REGION Network 3: ANGLE CODE READING
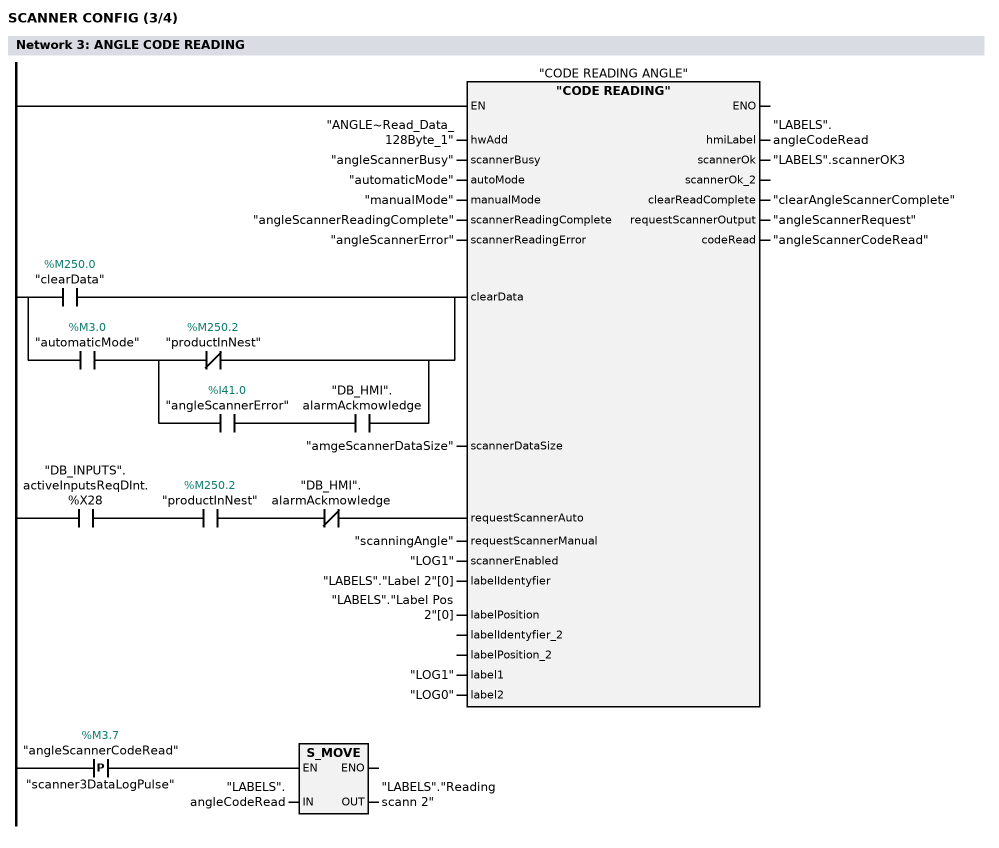
   RUNG wire#powerrail
      "CODE READING ANGLE"(clearData := wire#w2, requestScannerAuto := wire#w3, hwAdd := "ANGLE~Read_Data_128Byte_1", scannerBusy := "angleScannerBusy", autoMode := "automaticMode", manualMode := "manualMode", scannerReadingComplete := "angleScannerReadingComplete", scannerReadingError := "angleScannerError", scannerDataSize := "amgeScannerDataSize", requestScannerManual := "scanningAngle", scannerEnabled := "LOG1", labelIdentyfier := "LABELS"."Label 2"[0], labelPosition := "LABELS"."Label Pos 2"[0], labelIdentyfier_2 :=, labelPosition_2 :=, label1 := "LOG1", label2 := "LOG0", hmiLabel => "LABELS".angleCodeRead, scannerOk => "LABELS".scannerOK3, scannerOk_2 =>, clearReadComplete => "clearAngleScannerComplete", requestScannerOutput => "angleScannerRequest", codeRead => "angleScannerCodeRead")
   END_RUNG
   RUNG wire#powerrail
      Contact( "clearData" )
   END_RUNG wire#w2
   RUNG wire#powerrail
      Contact( "automaticMode" )
      wire#w1
      I_Contact( "productInNest" )
   END_RUNG wire#w2
   RUNG wire#w1
      Contact( "angleScannerError" )
      Contact( "DB_HMI".alarmAckmowledge )
   END_RUNG wire#w2
   RUNG wire#powerrail
      Contact( "DB_INPUTS".activeInputsReqDInt.%X28 )
      Contact( "productInNest" )
      I_Contact( "DB_HMI".alarmAckmowledge )
   END_RUNG wire#w3
   RUNG wire#powerrail
      P_Contact(operand := "angleScannerCodeRead", bit := "scanner3DataLogPulse")
      S_Move(in := "LABELS".angleCodeRead, out => "LABELS"."Reading scann 2")
   END_RUNG
   // the same network as SCL:
   "CODE READING ANGLE"(hwAdd := "ANGLE~Read_Data_128Byte_1",   // "CODE READING"
                        scannerBusy := "angleScannerBusy",
                        autoMode := "automaticMode",
                        manualMode := "manualMode",
                        scannerReadingComplete := "angleScannerReadingComplete",
                        scannerReadingError := "angleScannerError",
                        clearData := "clearData" OR ("automaticMode" AND (NOT "productInNest" OR ("angleScannerError" AND "DB_HMI".alarmAckmowledge))),
                        scannerDataSize := "amgeScannerDataSize",
                        requestScannerAuto := "DB_INPUTS".activeInputsReqDInt.%X28 AND "productInNest" AND NOT "DB_HMI".alarmAckmowledge,
                        requestScannerManual := "scanningAngle",
                        scannerEnabled := "LOG1",
                        labelIdentyfier := "LABELS"."Label 2"[0],
                        labelPosition := "LABELS"."Label Pos 2"[0],
                        label1 := "LOG1",
                        label2 := "LOG0",
                        hmiLabel => "LABELS".angleCodeRead,
                        scannerOk => "LABELS".scannerOK3,
                        clearReadComplete => "clearAngleScannerComplete",
                        requestScannerOutput => "angleScannerRequest",
                        codeRead => "angleScannerCodeRead");
   #_w1 := "angleScannerCodeRead" AND NOT "scanner3DataLogPulse";   // rising edge of "angleScannerCodeRead"
   "scanner3DataLogPulse" := "angleScannerCodeRead";
   IF #_w1 THEN "LABELS"."Reading scann 2" := "LABELS".angleCodeRead; END_IF;
END_REGION

REGION Network 4: Move values to HMI
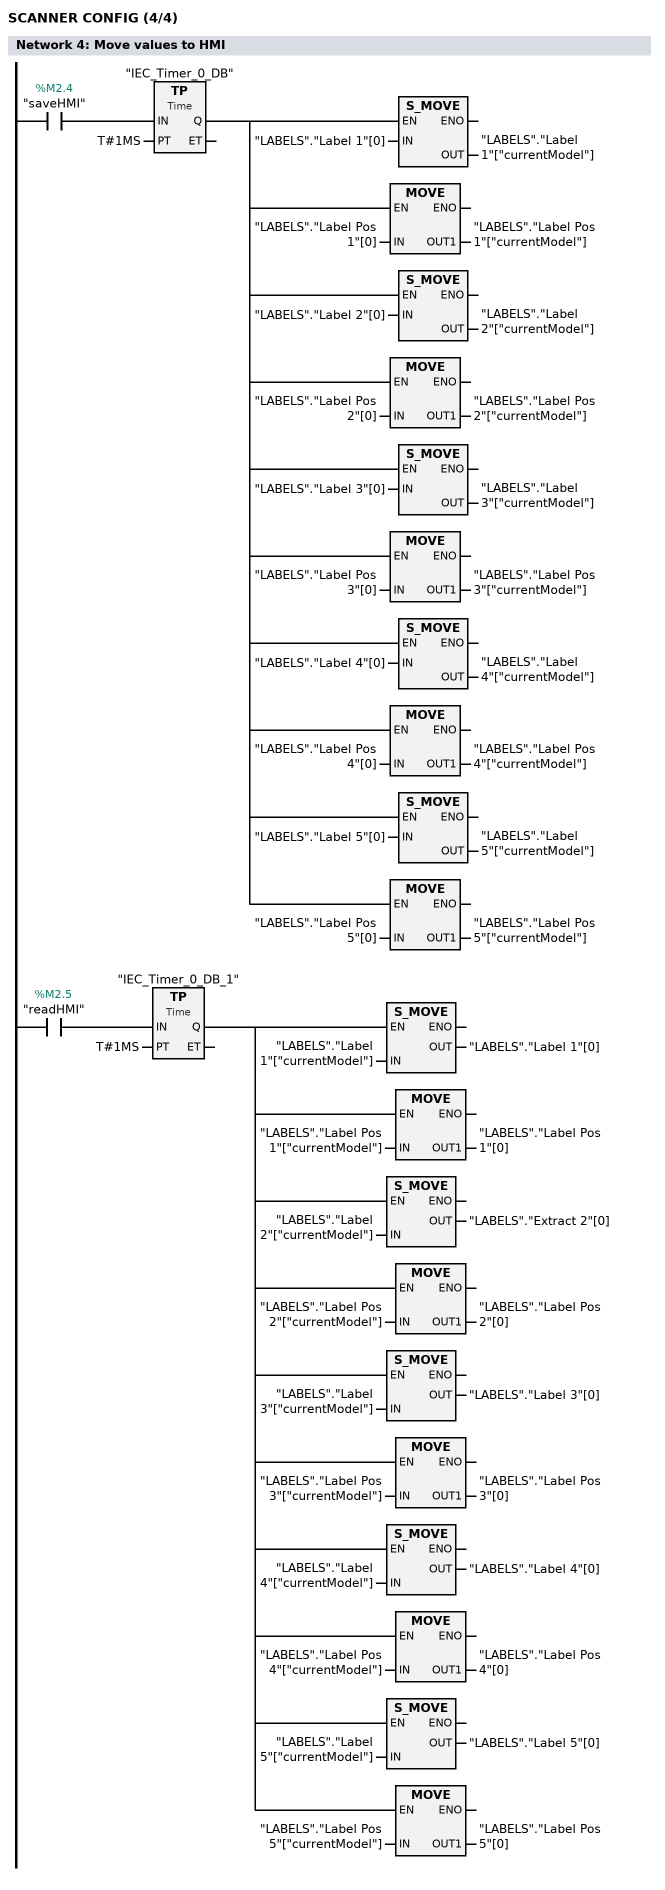
   RUNG wire#powerrail
      Contact( "saveHMI" )
      { S7_Templates := "time_type := Time" } "IEC_Timer_0_DB".TP(pt := T#1MS, et =>)
      wire#w1
      S_Move(in := "LABELS"."Label 1"[0], out => "LABELS"."Label 1"["currentModel"])
   END_RUNG
   RUNG wire#w1
      Move(in := "LABELS"."Label Pos 1"[0], out1 => "LABELS"."Label Pos 1"["currentModel"])
   END_RUNG
   RUNG wire#w1
      S_Move(in := "LABELS"."Label 2"[0], out => "LABELS"."Label 2"["currentModel"])
   END_RUNG
   RUNG wire#w1
      Move(in := "LABELS"."Label Pos 2"[0], out1 => "LABELS"."Label Pos 2"["currentModel"])
   END_RUNG
   RUNG wire#w1
      S_Move(in := "LABELS"."Label 3"[0], out => "LABELS"."Label 3"["currentModel"])
   END_RUNG
   RUNG wire#w1
      Move(in := "LABELS"."Label Pos 3"[0], out1 => "LABELS"."Label Pos 3"["currentModel"])
   END_RUNG
   RUNG wire#w1
      S_Move(in := "LABELS"."Label 4"[0], out => "LABELS"."Label 4"["currentModel"])
   END_RUNG
   RUNG wire#w1
      Move(in := "LABELS"."Label Pos 4"[0], out1 => "LABELS"."Label Pos 4"["currentModel"])
   END_RUNG
   RUNG wire#w1
      S_Move(in := "LABELS"."Label 5"[0], out => "LABELS"."Label 5"["currentModel"])
   END_RUNG
   RUNG wire#w1
      Move(in := "LABELS"."Label Pos 5"[0], out1 => "LABELS"."Label Pos 5"["currentModel"])
   END_RUNG
   RUNG wire#powerrail
      Contact( "readHMI" )
      { S7_Templates := "time_type := Time" } "IEC_Timer_0_DB_1".TP(pt := T#1MS, et =>)
      wire#w2
      S_Move(in := "LABELS"."Label 1"["currentModel"], out => "LABELS"."Label 1"[0])
   END_RUNG
   RUNG wire#w2
      Move(in := "LABELS"."Label Pos 1"["currentModel"], out1 => "LABELS"."Label Pos 1"[0])
   END_RUNG
   RUNG wire#w2
      S_Move(in := "LABELS"."Label 2"["currentModel"], out => "LABELS"."Extract 2"[0])
   END_RUNG
   RUNG wire#w2
      Move(in := "LABELS"."Label Pos 2"["currentModel"], out1 => "LABELS"."Label Pos 2"[0])
   END_RUNG
   RUNG wire#w2
      S_Move(in := "LABELS"."Label 3"["currentModel"], out => "LABELS"."Label 3"[0])
   END_RUNG
   RUNG wire#w2
      Move(in := "LABELS"."Label Pos 3"["currentModel"], out1 => "LABELS"."Label Pos 3"[0])
   END_RUNG
   RUNG wire#w2
      S_Move(in := "LABELS"."Label 4"["currentModel"], out => "LABELS"."Label 4"[0])
   END_RUNG
   RUNG wire#w2
      Move(in := "LABELS"."Label Pos 4"["currentModel"], out1 => "LABELS"."Label Pos 4"[0])
   END_RUNG
   RUNG wire#w2
      S_Move(in := "LABELS"."Label 5"["currentModel"], out => "LABELS"."Label 5"[0])
   END_RUNG
   RUNG wire#w2
      Move(in := "LABELS"."Label Pos 5"["currentModel"], out1 => "LABELS"."Label Pos 5"[0])
   END_RUNG
   // the same network as SCL:
   "IEC_Timer_0_DB".TP(IN := "saveHMI", PT := T#1MS);
   IF "IEC_Timer_0_DB".Q THEN
       "LABELS"."Label 1"["currentModel"] := "LABELS"."Label 1"[0];
       "LABELS"."Label Pos 1"["currentModel"] := "LABELS"."Label Pos 1"[0];
       "LABELS"."Label 2"["currentModel"] := "LABELS"."Label 2"[0];
       "LABELS"."Label Pos 2"["currentModel"] := "LABELS"."Label Pos 2"[0];
       "LABELS"."Label 3"["currentModel"] := "LABELS"."Label 3"[0];
       "LABELS"."Label Pos 3"["currentModel"] := "LABELS"."Label Pos 3"[0];
       "LABELS"."Label 4"["currentModel"] := "LABELS"."Label 4"[0];
       "LABELS"."Label Pos 4"["currentModel"] := "LABELS"."Label Pos 4"[0];
       "LABELS"."Label 5"["currentModel"] := "LABELS"."Label 5"[0];
       "LABELS"."Label Pos 5"["currentModel"] := "LABELS"."Label Pos 5"[0];
   END_IF;
   "IEC_Timer_0_DB_1".TP(IN := "readHMI", PT := T#1MS);
   IF "IEC_Timer_0_DB_1".Q THEN
       "LABELS"."Label 1"[0] := "LABELS"."Label 1"["currentModel"];
       "LABELS"."Label Pos 1"[0] := "LABELS"."Label Pos 1"["currentModel"];
       "LABELS"."Extract 2"[0] := "LABELS"."Label 2"["currentModel"];
       "LABELS"."Label Pos 2"[0] := "LABELS"."Label Pos 2"["currentModel"];
       "LABELS"."Label 3"[0] := "LABELS"."Label 3"["currentModel"];
       "LABELS"."Label Pos 3"[0] := "LABELS"."Label Pos 3"["currentModel"];
       "LABELS"."Label 4"[0] := "LABELS"."Label 4"["currentModel"];
       "LABELS"."Label Pos 4"[0] := "LABELS"."Label Pos 4"["currentModel"];
       "LABELS"."Label 5"[0] := "LABELS"."Label 5"["currentModel"];
       "LABELS"."Label Pos 5"[0] := "LABELS"."Label Pos 5"["currentModel"];
   END_IF;
END_REGION
END_FUNCTION

FUNCTION_BLOCK "CODE READING"   // FB13, LAD
{ S7_Optimized_Access := 'TRUE' }
VERSION : 0.1
// stored: AutoNumber true, IsIECCheckEnabled false, IsRetainMemResEnabled false, MemoryReserve 100, SetENOAutomatically false, UDAEnableTagReadback false
   VAR_INPUT
      hwAdd : HW_IO;
      scannerBusy : Bool;
      autoMode : Bool;
      manualMode : Bool;
      scannerReadingComplete : Bool;
      scannerReadingError : Bool;
      clearData : Bool;
      scannerDataSize : Int;
      requestScannerAuto : Bool;
      requestScannerManual : Bool;
      scannerEnabled : Bool;
      labelIdentyfier : String[5];
      labelPosition : Int;
      labelIdentyfier_2 : String[5];
      labelPosition_2 : Int;
      label1 : Bool;
      label2 : Bool;
   END_VAR
   VAR_OUTPUT
      hmiLabel : String[180];
      scannerOk : Bool;
      scannerOk_2 : Bool;
      clearReadComplete : Bool;
      requestScannerOutput : Bool;
      codeRead : Bool;
   END_VAR
   VAR
      scannerReading { ExternalAccessible := 'False'; ExternalVisible := 'False'; ExternalWritable := 'False'} : Array[0..254] of Char;
      ScannerReadTimer { S7_SetPoint := 'True'} : TON_TIME;
   END_VAR
   VAR_TEMP
      scannerError : Int;
      receiveCode : String[80];
      readingScann1 : String[180];
      scannerLength : Int;
      labelExtract : String[10];
   END_VAR
   VAR_TEMP   // added for the SCL form of the ladder/FBD networks
      _w1 : Bool;
      _w2 : Bool;
      _w3 : Bool;
      _w4 : Bool;
      _w5 : Bool;
      _w6 : Bool;
      _w7 : Bool;
      _w8 : Bool;
      _w9 : Bool;
      _w10 : Bool;
      _w11 : Bool;
   END_VAR
BEGIN

REGION Network 1: REQUEST SCANNER
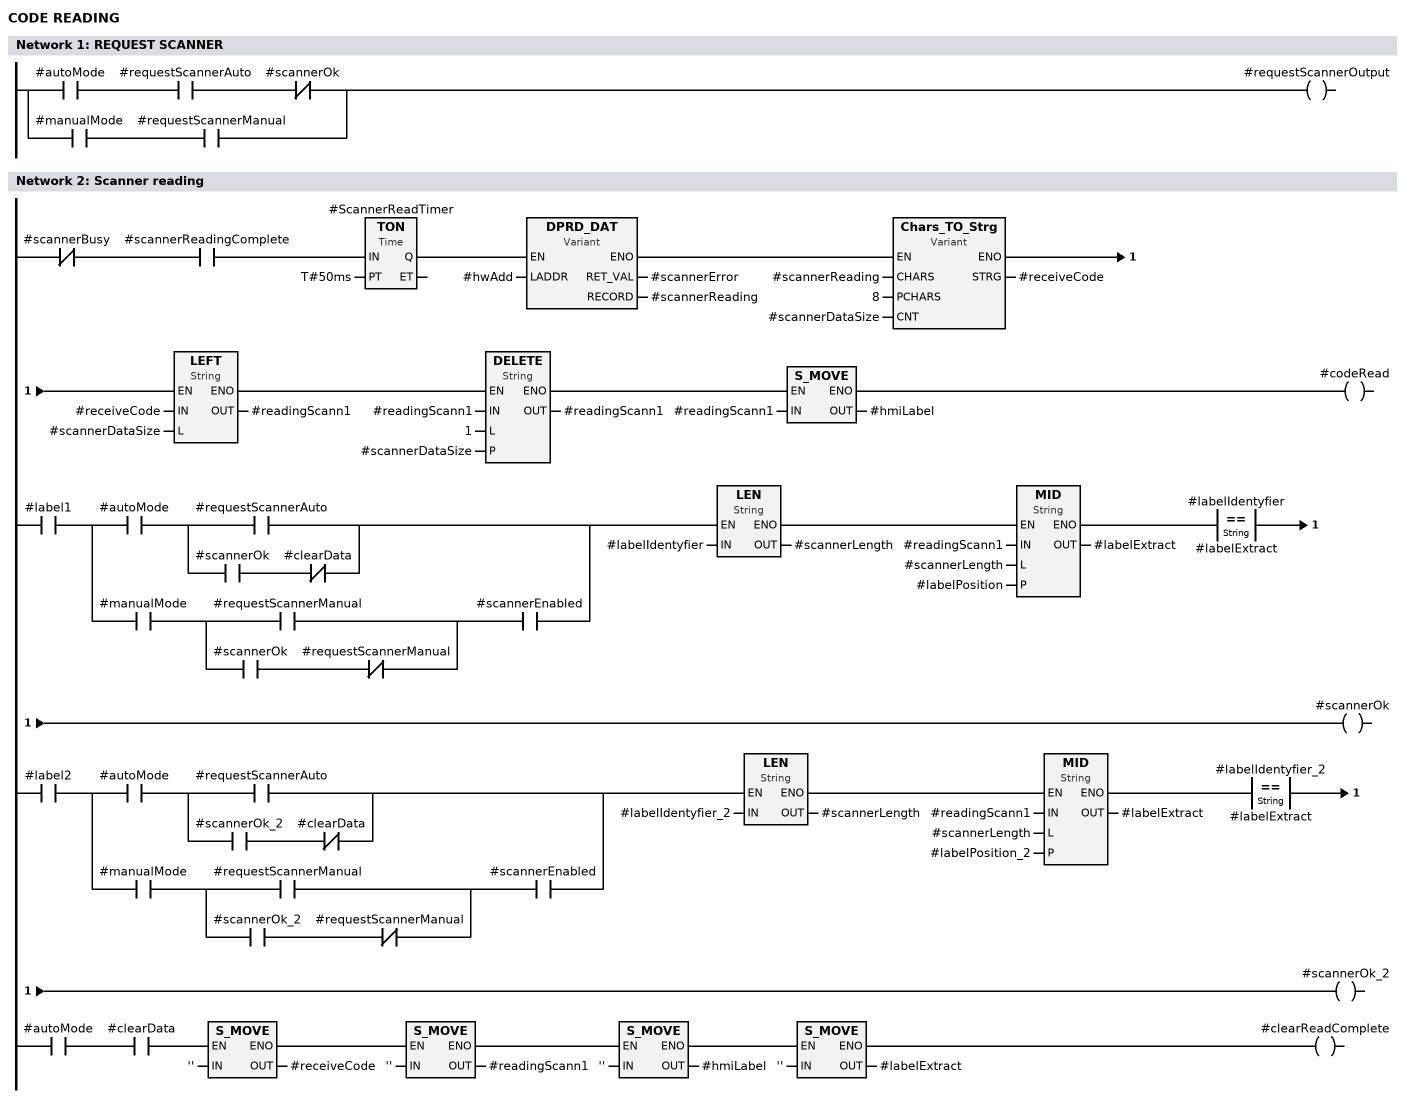
   RUNG wire#powerrail
      Contact( #autoMode )
      Contact( #requestScannerAuto )
      I_Contact( #scannerOk )
      wire#w1
      Coil( #requestScannerOutput )
   END_RUNG
   RUNG wire#powerrail
      Contact( #manualMode )
      Contact( #requestScannerManual )
   END_RUNG wire#w1
   // the same network as SCL:
   #requestScannerOutput := (#autoMode AND #requestScannerAuto AND NOT #scannerOk) OR (#manualMode AND #requestScannerManual);
END_REGION

REGION Network 2: Scanner reading
   RUNG wire#powerrail
      I_Contact( #scannerBusy )
      Contact( #scannerReadingComplete )
      { S7_Templates := "time_type := Time" } #ScannerReadTimer.TON(pt := T#50ms, et =>)
      { S7_Templates := "[ptr_type := Variant, laddr_type := HW_IO]" } DPRD_DAT(LADDR := #hwAdd, RET_VAL => #scannerError, RECORD => #scannerReading)
      { S7_Templates := "[ptr_type := Variant, str_type := String]" } Chars_TO_Strg(Chars := #scannerReading, pChars := 8, Cnt := #scannerDataSize, Strg => #receiveCode)
      { S7_Templates := "str_type := String" } LEFT(IN := #receiveCode, L := #scannerDataSize, OUT => #readingScann1)
      { S7_Templates := "str_type := String" } DELETE(IN := #readingScann1, L := 1, P := #scannerDataSize, OUT => #readingScann1)
      S_Move(in := #readingScann1, out => #hmiLabel)
      Coil( #codeRead )
   END_RUNG
   RUNG wire#powerrail
      Contact( #label1 )
      wire#w1
      Contact( #autoMode )
      wire#w2
      Contact( #requestScannerAuto )
      wire#w3
      { S7_Templates := "[str_type := String, return_type := Int]" } LEN(IN := #labelIdentyfier, OUT => #scannerLength)
      { S7_Templates := "value_type := String" } MID(IN := #readingScann1, L := #scannerLength, P := #labelPosition, OUT => #labelExtract)
      { S7_Templates := "SrcType := String" } EQ_Contact(in1 := #labelIdentyfier, in2 := #labelExtract)
      Coil( #scannerOk )
   END_RUNG
   RUNG wire#w2
      Contact( #scannerOk )
      I_Contact( #clearData )
   END_RUNG wire#w3
   RUNG wire#w1
      Contact( #manualMode )
      wire#w4
      Contact( #requestScannerManual )
      wire#w5
      Contact( #scannerEnabled )
   END_RUNG wire#w3
   RUNG wire#w4
      Contact( #scannerOk )
      I_Contact( #requestScannerManual )
   END_RUNG wire#w5
   RUNG wire#powerrail
      Contact( #label2 )
      wire#w6
      Contact( #autoMode )
      wire#w7
      Contact( #requestScannerAuto )
      wire#w8
      { S7_Templates := "[str_type := String, return_type := Int]" } LEN(IN := #labelIdentyfier_2, OUT => #scannerLength)
      { S7_Templates := "value_type := String" } MID(IN := #readingScann1, L := #scannerLength, P := #labelPosition_2, OUT => #labelExtract)
      { S7_Templates := "SrcType := String" } EQ_Contact(in1 := #labelIdentyfier_2, in2 := #labelExtract)
      Coil( #scannerOk_2 )
   END_RUNG
   RUNG wire#w7
      Contact( #scannerOk_2 )
      I_Contact( #clearData )
   END_RUNG wire#w8
   RUNG wire#w6
      Contact( #manualMode )
      wire#w9
      Contact( #requestScannerManual )
      wire#w10
      Contact( #scannerEnabled )
   END_RUNG wire#w8
   RUNG wire#w9
      Contact( #scannerOk_2 )
      I_Contact( #requestScannerManual )
   END_RUNG wire#w10
   RUNG wire#powerrail
      Contact( #autoMode )
      Contact( #clearData )
      S_Move(in := '', out => #receiveCode)
      S_Move(in := '', out => #readingScann1)
      S_Move(in := '', out => #hmiLabel)
      S_Move(in := '', out => #labelExtract)
      Coil( #clearReadComplete )
   END_RUNG
   // the same network as SCL:
   #ScannerReadTimer(IN := NOT #scannerBusy AND #scannerReadingComplete, PT := T#50ms);   // TON
   #scannerError := DPRD_DAT(EN := #ScannerReadTimer.Q, LADDR := #hwAdd, RECORD => #scannerReading, ENO => #_w1);
   Chars_TO_Strg(EN := #_w1,
                 Chars := #scannerReading,
                 pChars := 8,
                 Cnt := #scannerDataSize,
                 Strg => #receiveCode,
                 ENO => #_w2);
   LEFT(EN := #_w2, IN := #receiveCode, L := #scannerDataSize, OUT => #readingScann1, ENO => #_w3);
   DELETE(EN := #_w3, IN := #readingScann1, L := 1, P := #scannerDataSize, OUT => #readingScann1, ENO => #_w4);
   IF #_w4 THEN #hmiLabel := #readingScann1; END_IF;
   #codeRead := #_w4;
   #_w5 := #label1 AND ((#autoMode AND (#requestScannerAuto OR (#scannerOk AND NOT #clearData))) OR (#manualMode AND (#requestScannerManual OR (#scannerOk AND NOT #requestScannerManual)) AND #scannerEnabled));
   LEN(EN := #_w5, IN := #labelIdentyfier, OUT => #scannerLength, ENO => #_w6);
   MID(EN := #_w6,
       IN := #readingScann1,
       L := #scannerLength,
       P := #labelPosition,
       OUT => #labelExtract,
       ENO => #_w7);
   #scannerOk := #_w7 AND (#labelIdentyfier = #labelExtract);
   #_w8 := #label2 AND ((#autoMode AND (#requestScannerAuto OR (#scannerOk_2 AND NOT #clearData))) OR (#manualMode AND (#requestScannerManual OR (#scannerOk_2 AND NOT #requestScannerManual)) AND #scannerEnabled));
   LEN(EN := #_w8, IN := #labelIdentyfier_2, OUT => #scannerLength, ENO => #_w9);
   MID(EN := #_w9,
       IN := #readingScann1,
       L := #scannerLength,
       P := #labelPosition_2,
       OUT => #labelExtract,
       ENO => #_w10);
   #scannerOk_2 := #_w10 AND (#labelIdentyfier_2 = #labelExtract);
   #_w11 := #autoMode AND #clearData;
   IF #_w11 THEN
       #receiveCode := '';
       #readingScann1 := '';
       #hmiLabel := '';
       #labelExtract := '';
   END_IF;
   #clearReadComplete := #_w11;
END_REGION
END_FUNCTION_BLOCK

FUNCTION "DINT TO BOOL" : Void   // FC10, LAD
{ S7_Optimized_Access := 'TRUE' }
VERSION : 0.1
// stored: AutoNumber true, IsIECCheckEnabled false, SetENOAutomatically false, UDAEnableTagReadback false
BEGIN

REGION Network 1: A INPUTS STATUS
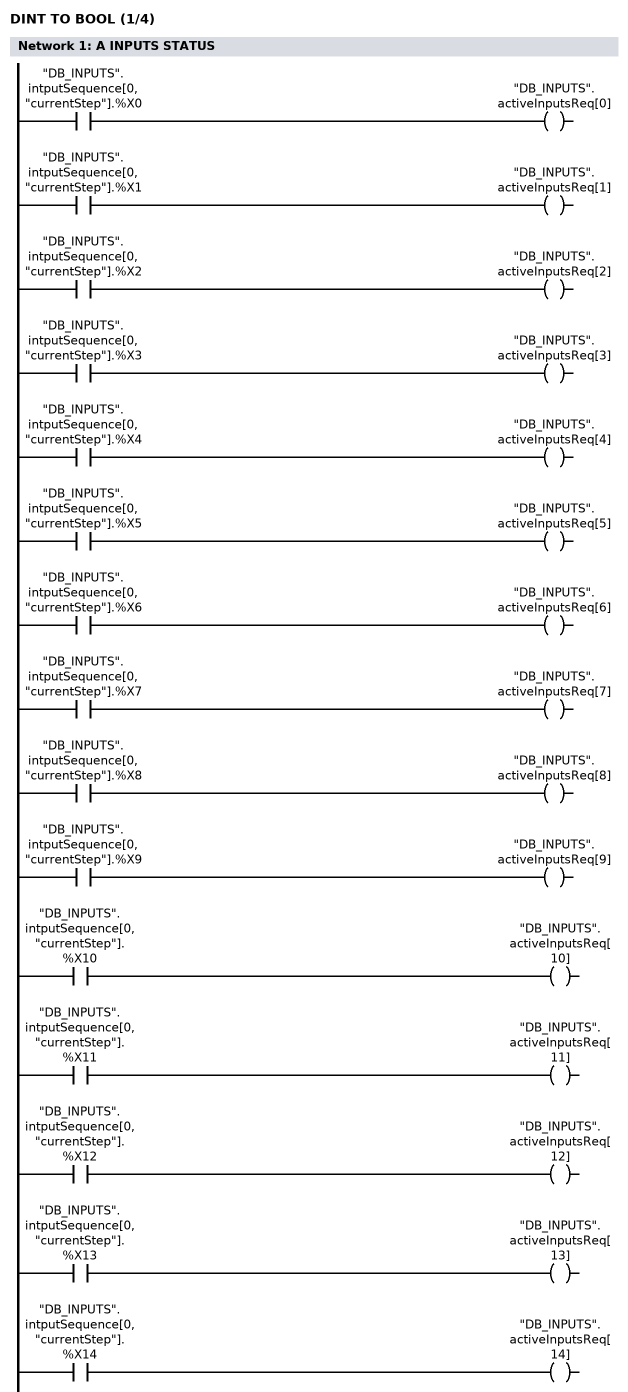
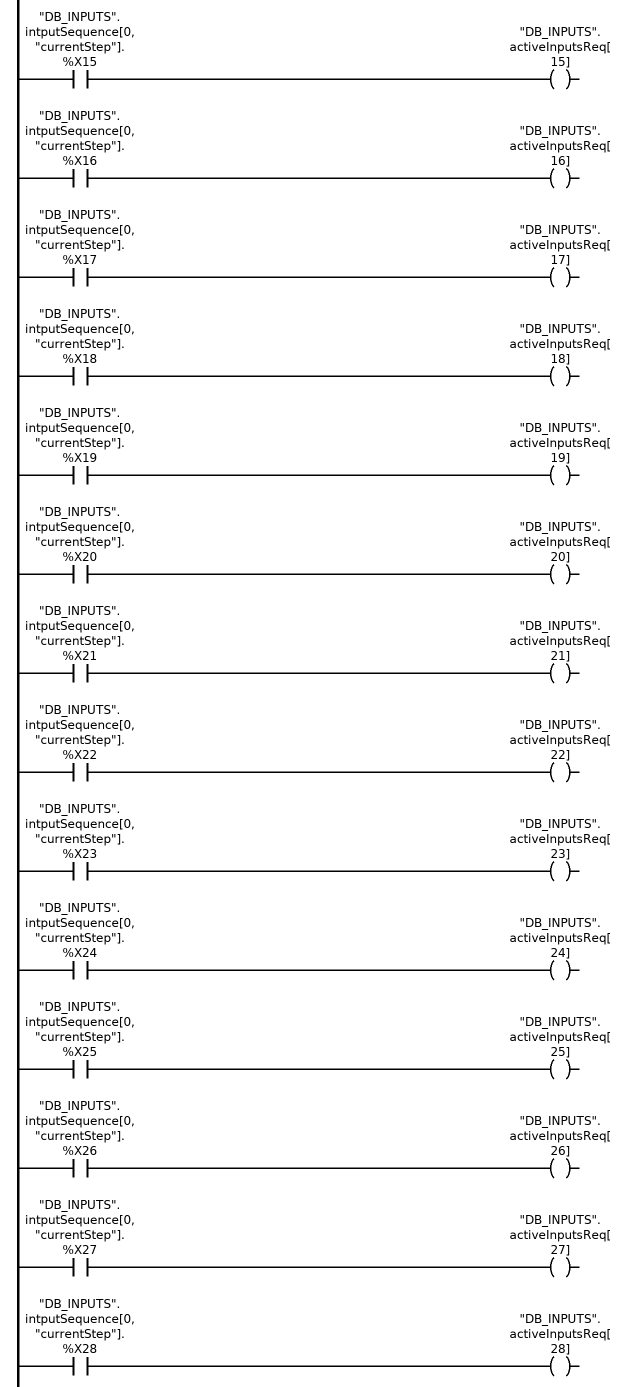
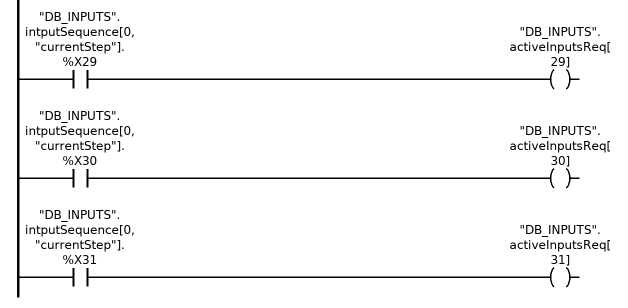
   RUNG wire#powerrail
      Contact( "DB_INPUTS".intputSequence[0, "currentStep"].%X0 )
      Coil( "DB_INPUTS".activeInputsReq[0] )
   END_RUNG
   RUNG wire#powerrail
      Contact( "DB_INPUTS".intputSequence[0, "currentStep"].%X1 )
      Coil( "DB_INPUTS".activeInputsReq[1] )
   END_RUNG
   RUNG wire#powerrail
      Contact( "DB_INPUTS".intputSequence[0, "currentStep"].%X2 )
      Coil( "DB_INPUTS".activeInputsReq[2] )
   END_RUNG
   RUNG wire#powerrail
      Contact( "DB_INPUTS".intputSequence[0, "currentStep"].%X3 )
      Coil( "DB_INPUTS".activeInputsReq[3] )
   END_RUNG
   RUNG wire#powerrail
      Contact( "DB_INPUTS".intputSequence[0, "currentStep"].%X4 )
      Coil( "DB_INPUTS".activeInputsReq[4] )
   END_RUNG
   RUNG wire#powerrail
      Contact( "DB_INPUTS".intputSequence[0, "currentStep"].%X5 )
      Coil( "DB_INPUTS".activeInputsReq[5] )
   END_RUNG
   RUNG wire#powerrail
      Contact( "DB_INPUTS".intputSequence[0, "currentStep"].%X6 )
      Coil( "DB_INPUTS".activeInputsReq[6] )
   END_RUNG
   RUNG wire#powerrail
      Contact( "DB_INPUTS".intputSequence[0, "currentStep"].%X7 )
      Coil( "DB_INPUTS".activeInputsReq[7] )
   END_RUNG
   RUNG wire#powerrail
      Contact( "DB_INPUTS".intputSequence[0, "currentStep"].%X8 )
      Coil( "DB_INPUTS".activeInputsReq[8] )
   END_RUNG
   RUNG wire#powerrail
      Contact( "DB_INPUTS".intputSequence[0, "currentStep"].%X9 )
      Coil( "DB_INPUTS".activeInputsReq[9] )
   END_RUNG
   RUNG wire#powerrail
      Contact( "DB_INPUTS".intputSequence[0, "currentStep"].%X10 )
      Coil( "DB_INPUTS".activeInputsReq[10] )
   END_RUNG
   RUNG wire#powerrail
      Contact( "DB_INPUTS".intputSequence[0, "currentStep"].%X11 )
      Coil( "DB_INPUTS".activeInputsReq[11] )
   END_RUNG
   RUNG wire#powerrail
      Contact( "DB_INPUTS".intputSequence[0, "currentStep"].%X12 )
      Coil( "DB_INPUTS".activeInputsReq[12] )
   END_RUNG
   RUNG wire#powerrail
      Contact( "DB_INPUTS".intputSequence[0, "currentStep"].%X13 )
      Coil( "DB_INPUTS".activeInputsReq[13] )
   END_RUNG
   RUNG wire#powerrail
      Contact( "DB_INPUTS".intputSequence[0, "currentStep"].%X14 )
      Coil( "DB_INPUTS".activeInputsReq[14] )
   END_RUNG
   RUNG wire#powerrail
      Contact( "DB_INPUTS".intputSequence[0, "currentStep"].%X15 )
      Coil( "DB_INPUTS".activeInputsReq[15] )
   END_RUNG
   RUNG wire#powerrail
      Contact( "DB_INPUTS".intputSequence[0, "currentStep"].%X16 )
      Coil( "DB_INPUTS".activeInputsReq[16] )
   END_RUNG
   RUNG wire#powerrail
      Contact( "DB_INPUTS".intputSequence[0, "currentStep"].%X17 )
      Coil( "DB_INPUTS".activeInputsReq[17] )
   END_RUNG
   RUNG wire#powerrail
      Contact( "DB_INPUTS".intputSequence[0, "currentStep"].%X18 )
      Coil( "DB_INPUTS".activeInputsReq[18] )
   END_RUNG
   RUNG wire#powerrail
      Contact( "DB_INPUTS".intputSequence[0, "currentStep"].%X19 )
      Coil( "DB_INPUTS".activeInputsReq[19] )
   END_RUNG
   RUNG wire#powerrail
      Contact( "DB_INPUTS".intputSequence[0, "currentStep"].%X20 )
      Coil( "DB_INPUTS".activeInputsReq[20] )
   END_RUNG
   RUNG wire#powerrail
      Contact( "DB_INPUTS".intputSequence[0, "currentStep"].%X21 )
      Coil( "DB_INPUTS".activeInputsReq[21] )
   END_RUNG
   RUNG wire#powerrail
      Contact( "DB_INPUTS".intputSequence[0, "currentStep"].%X22 )
      Coil( "DB_INPUTS".activeInputsReq[22] )
   END_RUNG
   RUNG wire#powerrail
      Contact( "DB_INPUTS".intputSequence[0, "currentStep"].%X23 )
      Coil( "DB_INPUTS".activeInputsReq[23] )
   END_RUNG
   RUNG wire#powerrail
      Contact( "DB_INPUTS".intputSequence[0, "currentStep"].%X24 )
      Coil( "DB_INPUTS".activeInputsReq[24] )
   END_RUNG
   RUNG wire#powerrail
      Contact( "DB_INPUTS".intputSequence[0, "currentStep"].%X25 )
      Coil( "DB_INPUTS".activeInputsReq[25] )
   END_RUNG
   RUNG wire#powerrail
      Contact( "DB_INPUTS".intputSequence[0, "currentStep"].%X26 )
      Coil( "DB_INPUTS".activeInputsReq[26] )
   END_RUNG
   RUNG wire#powerrail
      Contact( "DB_INPUTS".intputSequence[0, "currentStep"].%X27 )
      Coil( "DB_INPUTS".activeInputsReq[27] )
   END_RUNG
   RUNG wire#powerrail
      Contact( "DB_INPUTS".intputSequence[0, "currentStep"].%X28 )
      Coil( "DB_INPUTS".activeInputsReq[28] )
   END_RUNG
   RUNG wire#powerrail
      Contact( "DB_INPUTS".intputSequence[0, "currentStep"].%X29 )
      Coil( "DB_INPUTS".activeInputsReq[29] )
   END_RUNG
   RUNG wire#powerrail
      Contact( "DB_INPUTS".intputSequence[0, "currentStep"].%X30 )
      Coil( "DB_INPUTS".activeInputsReq[30] )
   END_RUNG
   RUNG wire#powerrail
      Contact( "DB_INPUTS".intputSequence[0, "currentStep"].%X31 )
      Coil( "DB_INPUTS".activeInputsReq[31] )
   END_RUNG
   // the same network as SCL:
   "DB_INPUTS".activeInputsReq[0] := "DB_INPUTS".intputSequence[0, "currentStep"].%X0;
   "DB_INPUTS".activeInputsReq[1] := "DB_INPUTS".intputSequence[0, "currentStep"].%X1;
   "DB_INPUTS".activeInputsReq[2] := "DB_INPUTS".intputSequence[0, "currentStep"].%X2;
   "DB_INPUTS".activeInputsReq[3] := "DB_INPUTS".intputSequence[0, "currentStep"].%X3;
   "DB_INPUTS".activeInputsReq[4] := "DB_INPUTS".intputSequence[0, "currentStep"].%X4;
   "DB_INPUTS".activeInputsReq[5] := "DB_INPUTS".intputSequence[0, "currentStep"].%X5;
   "DB_INPUTS".activeInputsReq[6] := "DB_INPUTS".intputSequence[0, "currentStep"].%X6;
   "DB_INPUTS".activeInputsReq[7] := "DB_INPUTS".intputSequence[0, "currentStep"].%X7;
   "DB_INPUTS".activeInputsReq[8] := "DB_INPUTS".intputSequence[0, "currentStep"].%X8;
   "DB_INPUTS".activeInputsReq[9] := "DB_INPUTS".intputSequence[0, "currentStep"].%X9;
   "DB_INPUTS".activeInputsReq[10] := "DB_INPUTS".intputSequence[0, "currentStep"].%X10;
   "DB_INPUTS".activeInputsReq[11] := "DB_INPUTS".intputSequence[0, "currentStep"].%X11;
   "DB_INPUTS".activeInputsReq[12] := "DB_INPUTS".intputSequence[0, "currentStep"].%X12;
   "DB_INPUTS".activeInputsReq[13] := "DB_INPUTS".intputSequence[0, "currentStep"].%X13;
   "DB_INPUTS".activeInputsReq[14] := "DB_INPUTS".intputSequence[0, "currentStep"].%X14;
   "DB_INPUTS".activeInputsReq[15] := "DB_INPUTS".intputSequence[0, "currentStep"].%X15;
   "DB_INPUTS".activeInputsReq[16] := "DB_INPUTS".intputSequence[0, "currentStep"].%X16;
   "DB_INPUTS".activeInputsReq[17] := "DB_INPUTS".intputSequence[0, "currentStep"].%X17;
   "DB_INPUTS".activeInputsReq[18] := "DB_INPUTS".intputSequence[0, "currentStep"].%X18;
   "DB_INPUTS".activeInputsReq[19] := "DB_INPUTS".intputSequence[0, "currentStep"].%X19;
   "DB_INPUTS".activeInputsReq[20] := "DB_INPUTS".intputSequence[0, "currentStep"].%X20;
   "DB_INPUTS".activeInputsReq[21] := "DB_INPUTS".intputSequence[0, "currentStep"].%X21;
   "DB_INPUTS".activeInputsReq[22] := "DB_INPUTS".intputSequence[0, "currentStep"].%X22;
   "DB_INPUTS".activeInputsReq[23] := "DB_INPUTS".intputSequence[0, "currentStep"].%X23;
   "DB_INPUTS".activeInputsReq[24] := "DB_INPUTS".intputSequence[0, "currentStep"].%X24;
   "DB_INPUTS".activeInputsReq[25] := "DB_INPUTS".intputSequence[0, "currentStep"].%X25;
   "DB_INPUTS".activeInputsReq[26] := "DB_INPUTS".intputSequence[0, "currentStep"].%X26;
   "DB_INPUTS".activeInputsReq[27] := "DB_INPUTS".intputSequence[0, "currentStep"].%X27;
   "DB_INPUTS".activeInputsReq[28] := "DB_INPUTS".intputSequence[0, "currentStep"].%X28;
   "DB_INPUTS".activeInputsReq[29] := "DB_INPUTS".intputSequence[0, "currentStep"].%X29;
   "DB_INPUTS".activeInputsReq[30] := "DB_INPUTS".intputSequence[0, "currentStep"].%X30;
   "DB_INPUTS".activeInputsReq[31] := "DB_INPUTS".intputSequence[0, "currentStep"].%X31;
END_REGION

REGION Network 2: MASK INPUTS STATUS
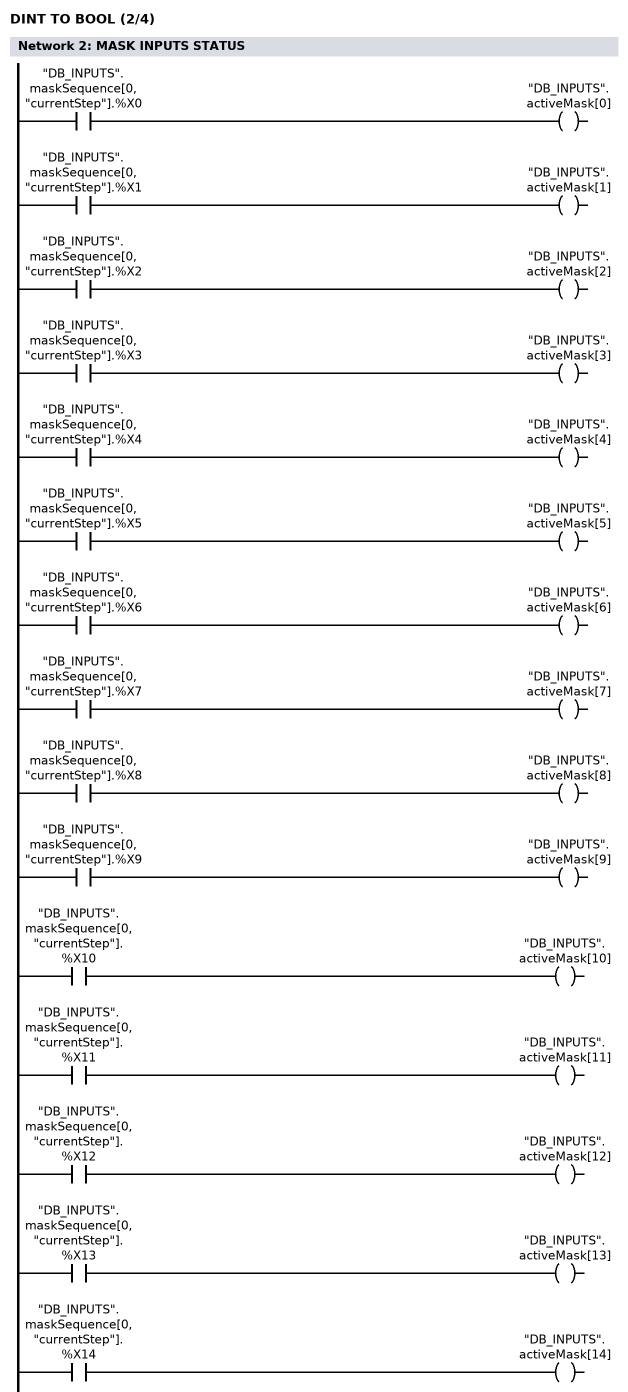
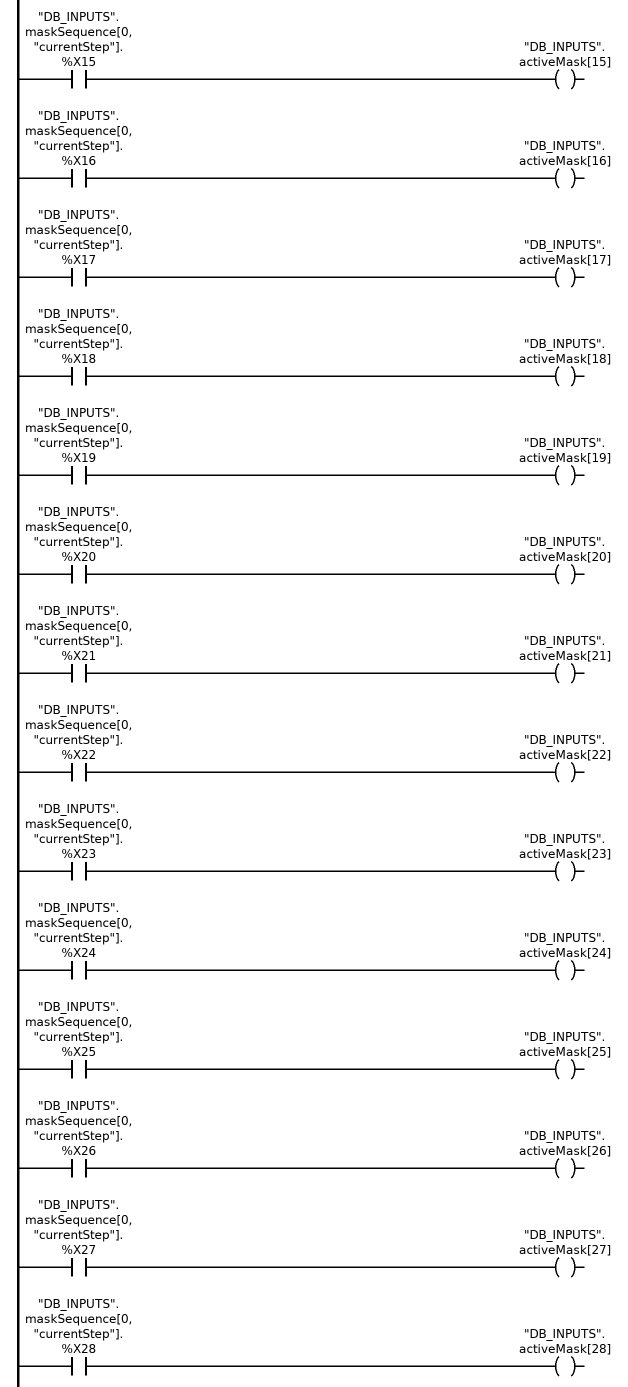
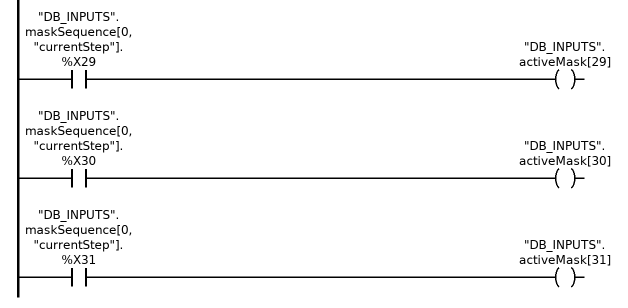
   RUNG wire#powerrail
      Contact( "DB_INPUTS".maskSequence[0, "currentStep"].%X0 )
      Coil( "DB_INPUTS".activeMask[0] )
   END_RUNG
   RUNG wire#powerrail
      Contact( "DB_INPUTS".maskSequence[0, "currentStep"].%X1 )
      Coil( "DB_INPUTS".activeMask[1] )
   END_RUNG
   RUNG wire#powerrail
      Contact( "DB_INPUTS".maskSequence[0, "currentStep"].%X2 )
      Coil( "DB_INPUTS".activeMask[2] )
   END_RUNG
   RUNG wire#powerrail
      Contact( "DB_INPUTS".maskSequence[0, "currentStep"].%X3 )
      Coil( "DB_INPUTS".activeMask[3] )
   END_RUNG
   RUNG wire#powerrail
      Contact( "DB_INPUTS".maskSequence[0, "currentStep"].%X4 )
      Coil( "DB_INPUTS".activeMask[4] )
   END_RUNG
   RUNG wire#powerrail
      Contact( "DB_INPUTS".maskSequence[0, "currentStep"].%X5 )
      Coil( "DB_INPUTS".activeMask[5] )
   END_RUNG
   RUNG wire#powerrail
      Contact( "DB_INPUTS".maskSequence[0, "currentStep"].%X6 )
      Coil( "DB_INPUTS".activeMask[6] )
   END_RUNG
   RUNG wire#powerrail
      Contact( "DB_INPUTS".maskSequence[0, "currentStep"].%X7 )
      Coil( "DB_INPUTS".activeMask[7] )
   END_RUNG
   RUNG wire#powerrail
      Contact( "DB_INPUTS".maskSequence[0, "currentStep"].%X8 )
      Coil( "DB_INPUTS".activeMask[8] )
   END_RUNG
   RUNG wire#powerrail
      Contact( "DB_INPUTS".maskSequence[0, "currentStep"].%X9 )
      Coil( "DB_INPUTS".activeMask[9] )
   END_RUNG
   RUNG wire#powerrail
      Contact( "DB_INPUTS".maskSequence[0, "currentStep"].%X10 )
      Coil( "DB_INPUTS".activeMask[10] )
   END_RUNG
   RUNG wire#powerrail
      Contact( "DB_INPUTS".maskSequence[0, "currentStep"].%X11 )
      Coil( "DB_INPUTS".activeMask[11] )
   END_RUNG
   RUNG wire#powerrail
      Contact( "DB_INPUTS".maskSequence[0, "currentStep"].%X12 )
      Coil( "DB_INPUTS".activeMask[12] )
   END_RUNG
   RUNG wire#powerrail
      Contact( "DB_INPUTS".maskSequence[0, "currentStep"].%X13 )
      Coil( "DB_INPUTS".activeMask[13] )
   END_RUNG
   RUNG wire#powerrail
      Contact( "DB_INPUTS".maskSequence[0, "currentStep"].%X14 )
      Coil( "DB_INPUTS".activeMask[14] )
   END_RUNG
   RUNG wire#powerrail
      Contact( "DB_INPUTS".maskSequence[0, "currentStep"].%X15 )
      Coil( "DB_INPUTS".activeMask[15] )
   END_RUNG
   RUNG wire#powerrail
      Contact( "DB_INPUTS".maskSequence[0, "currentStep"].%X16 )
      Coil( "DB_INPUTS".activeMask[16] )
   END_RUNG
   RUNG wire#powerrail
      Contact( "DB_INPUTS".maskSequence[0, "currentStep"].%X17 )
      Coil( "DB_INPUTS".activeMask[17] )
   END_RUNG
   RUNG wire#powerrail
      Contact( "DB_INPUTS".maskSequence[0, "currentStep"].%X18 )
      Coil( "DB_INPUTS".activeMask[18] )
   END_RUNG
   RUNG wire#powerrail
      Contact( "DB_INPUTS".maskSequence[0, "currentStep"].%X19 )
      Coil( "DB_INPUTS".activeMask[19] )
   END_RUNG
   RUNG wire#powerrail
      Contact( "DB_INPUTS".maskSequence[0, "currentStep"].%X20 )
      Coil( "DB_INPUTS".activeMask[20] )
   END_RUNG
   RUNG wire#powerrail
      Contact( "DB_INPUTS".maskSequence[0, "currentStep"].%X21 )
      Coil( "DB_INPUTS".activeMask[21] )
   END_RUNG
   RUNG wire#powerrail
      Contact( "DB_INPUTS".maskSequence[0, "currentStep"].%X22 )
      Coil( "DB_INPUTS".activeMask[22] )
   END_RUNG
   RUNG wire#powerrail
      Contact( "DB_INPUTS".maskSequence[0, "currentStep"].%X23 )
      Coil( "DB_INPUTS".activeMask[23] )
   END_RUNG
   RUNG wire#powerrail
      Contact( "DB_INPUTS".maskSequence[0, "currentStep"].%X24 )
      Coil( "DB_INPUTS".activeMask[24] )
   END_RUNG
   RUNG wire#powerrail
      Contact( "DB_INPUTS".maskSequence[0, "currentStep"].%X25 )
      Coil( "DB_INPUTS".activeMask[25] )
   END_RUNG
   RUNG wire#powerrail
      Contact( "DB_INPUTS".maskSequence[0, "currentStep"].%X26 )
      Coil( "DB_INPUTS".activeMask[26] )
   END_RUNG
   RUNG wire#powerrail
      Contact( "DB_INPUTS".maskSequence[0, "currentStep"].%X27 )
      Coil( "DB_INPUTS".activeMask[27] )
   END_RUNG
   RUNG wire#powerrail
      Contact( "DB_INPUTS".maskSequence[0, "currentStep"].%X28 )
      Coil( "DB_INPUTS".activeMask[28] )
   END_RUNG
   RUNG wire#powerrail
      Contact( "DB_INPUTS".maskSequence[0, "currentStep"].%X29 )
      Coil( "DB_INPUTS".activeMask[29] )
   END_RUNG
   RUNG wire#powerrail
      Contact( "DB_INPUTS".maskSequence[0, "currentStep"].%X30 )
      Coil( "DB_INPUTS".activeMask[30] )
   END_RUNG
   RUNG wire#powerrail
      Contact( "DB_INPUTS".maskSequence[0, "currentStep"].%X31 )
      Coil( "DB_INPUTS".activeMask[31] )
   END_RUNG
   // the same network as SCL:
   "DB_INPUTS".activeMask[0] := "DB_INPUTS".maskSequence[0, "currentStep"].%X0;
   "DB_INPUTS".activeMask[1] := "DB_INPUTS".maskSequence[0, "currentStep"].%X1;
   "DB_INPUTS".activeMask[2] := "DB_INPUTS".maskSequence[0, "currentStep"].%X2;
   "DB_INPUTS".activeMask[3] := "DB_INPUTS".maskSequence[0, "currentStep"].%X3;
   "DB_INPUTS".activeMask[4] := "DB_INPUTS".maskSequence[0, "currentStep"].%X4;
   "DB_INPUTS".activeMask[5] := "DB_INPUTS".maskSequence[0, "currentStep"].%X5;
   "DB_INPUTS".activeMask[6] := "DB_INPUTS".maskSequence[0, "currentStep"].%X6;
   "DB_INPUTS".activeMask[7] := "DB_INPUTS".maskSequence[0, "currentStep"].%X7;
   "DB_INPUTS".activeMask[8] := "DB_INPUTS".maskSequence[0, "currentStep"].%X8;
   "DB_INPUTS".activeMask[9] := "DB_INPUTS".maskSequence[0, "currentStep"].%X9;
   "DB_INPUTS".activeMask[10] := "DB_INPUTS".maskSequence[0, "currentStep"].%X10;
   "DB_INPUTS".activeMask[11] := "DB_INPUTS".maskSequence[0, "currentStep"].%X11;
   "DB_INPUTS".activeMask[12] := "DB_INPUTS".maskSequence[0, "currentStep"].%X12;
   "DB_INPUTS".activeMask[13] := "DB_INPUTS".maskSequence[0, "currentStep"].%X13;
   "DB_INPUTS".activeMask[14] := "DB_INPUTS".maskSequence[0, "currentStep"].%X14;
   "DB_INPUTS".activeMask[15] := "DB_INPUTS".maskSequence[0, "currentStep"].%X15;
   "DB_INPUTS".activeMask[16] := "DB_INPUTS".maskSequence[0, "currentStep"].%X16;
   "DB_INPUTS".activeMask[17] := "DB_INPUTS".maskSequence[0, "currentStep"].%X17;
   "DB_INPUTS".activeMask[18] := "DB_INPUTS".maskSequence[0, "currentStep"].%X18;
   "DB_INPUTS".activeMask[19] := "DB_INPUTS".maskSequence[0, "currentStep"].%X19;
   "DB_INPUTS".activeMask[20] := "DB_INPUTS".maskSequence[0, "currentStep"].%X20;
   "DB_INPUTS".activeMask[21] := "DB_INPUTS".maskSequence[0, "currentStep"].%X21;
   "DB_INPUTS".activeMask[22] := "DB_INPUTS".maskSequence[0, "currentStep"].%X22;
   "DB_INPUTS".activeMask[23] := "DB_INPUTS".maskSequence[0, "currentStep"].%X23;
   "DB_INPUTS".activeMask[24] := "DB_INPUTS".maskSequence[0, "currentStep"].%X24;
   "DB_INPUTS".activeMask[25] := "DB_INPUTS".maskSequence[0, "currentStep"].%X25;
   "DB_INPUTS".activeMask[26] := "DB_INPUTS".maskSequence[0, "currentStep"].%X26;
   "DB_INPUTS".activeMask[27] := "DB_INPUTS".maskSequence[0, "currentStep"].%X27;
   "DB_INPUTS".activeMask[28] := "DB_INPUTS".maskSequence[0, "currentStep"].%X28;
   "DB_INPUTS".activeMask[29] := "DB_INPUTS".maskSequence[0, "currentStep"].%X29;
   "DB_INPUTS".activeMask[30] := "DB_INPUTS".maskSequence[0, "currentStep"].%X30;
   "DB_INPUTS".activeMask[31] := "DB_INPUTS".maskSequence[0, "currentStep"].%X31;
END_REGION

REGION Network 3: B OUTPUTS STATUS
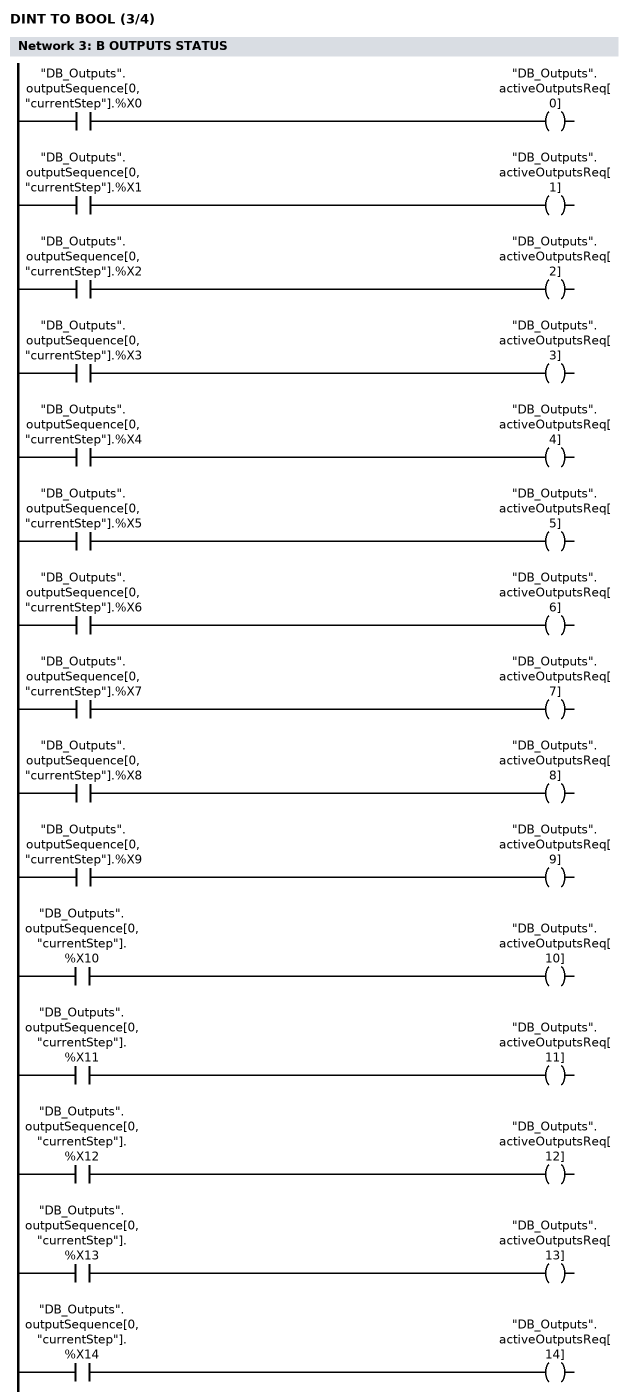
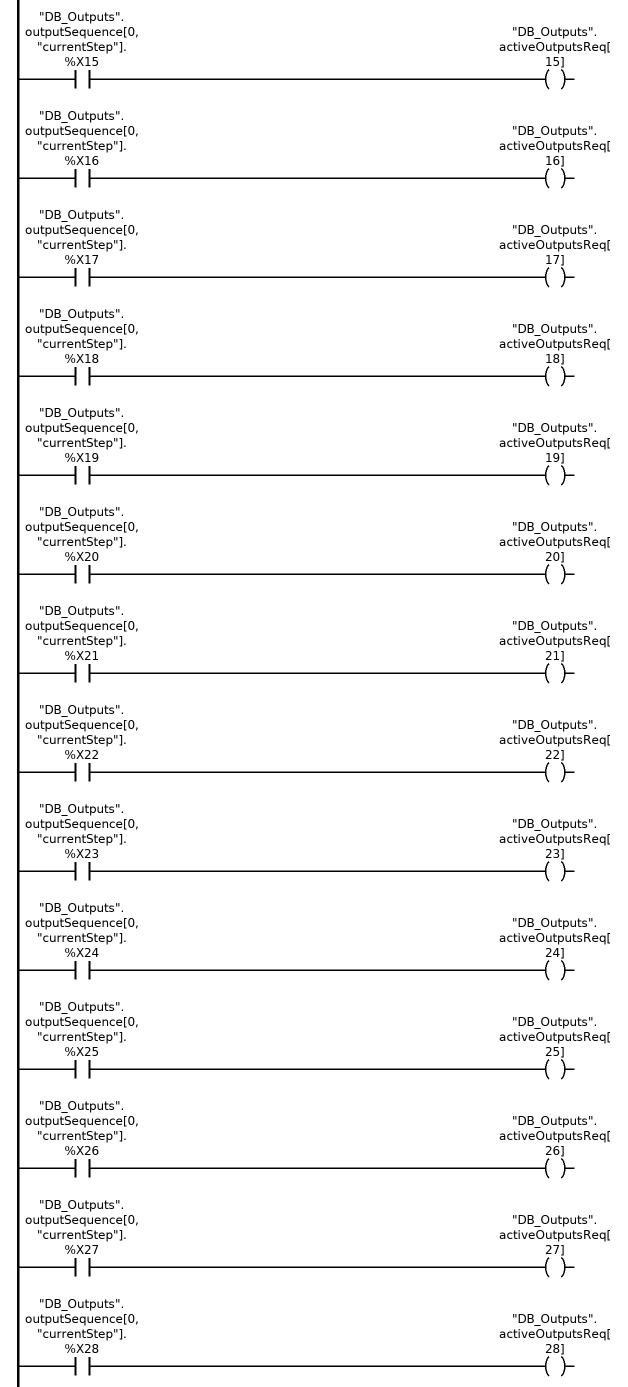
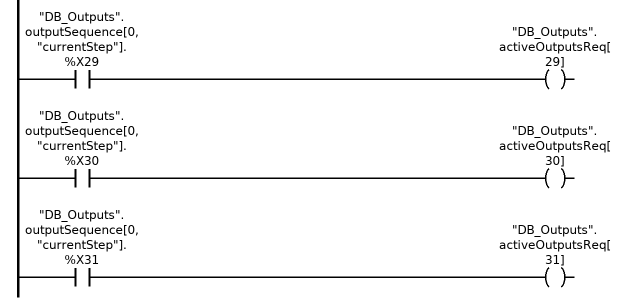
   RUNG wire#powerrail
      Contact( "DB_Outputs".outputSequence[0, "currentStep"].%X0 )
      Coil( "DB_Outputs".activeOutputsReq[0] )
   END_RUNG
   RUNG wire#powerrail
      Contact( "DB_Outputs".outputSequence[0, "currentStep"].%X1 )
      Coil( "DB_Outputs".activeOutputsReq[1] )
   END_RUNG
   RUNG wire#powerrail
      Contact( "DB_Outputs".outputSequence[0, "currentStep"].%X2 )
      Coil( "DB_Outputs".activeOutputsReq[2] )
   END_RUNG
   RUNG wire#powerrail
      Contact( "DB_Outputs".outputSequence[0, "currentStep"].%X3 )
      Coil( "DB_Outputs".activeOutputsReq[3] )
   END_RUNG
   RUNG wire#powerrail
      Contact( "DB_Outputs".outputSequence[0, "currentStep"].%X4 )
      Coil( "DB_Outputs".activeOutputsReq[4] )
   END_RUNG
   RUNG wire#powerrail
      Contact( "DB_Outputs".outputSequence[0, "currentStep"].%X5 )
      Coil( "DB_Outputs".activeOutputsReq[5] )
   END_RUNG
   RUNG wire#powerrail
      Contact( "DB_Outputs".outputSequence[0, "currentStep"].%X6 )
      Coil( "DB_Outputs".activeOutputsReq[6] )
   END_RUNG
   RUNG wire#powerrail
      Contact( "DB_Outputs".outputSequence[0, "currentStep"].%X7 )
      Coil( "DB_Outputs".activeOutputsReq[7] )
   END_RUNG
   RUNG wire#powerrail
      Contact( "DB_Outputs".outputSequence[0, "currentStep"].%X8 )
      Coil( "DB_Outputs".activeOutputsReq[8] )
   END_RUNG
   RUNG wire#powerrail
      Contact( "DB_Outputs".outputSequence[0, "currentStep"].%X9 )
      Coil( "DB_Outputs".activeOutputsReq[9] )
   END_RUNG
   RUNG wire#powerrail
      Contact( "DB_Outputs".outputSequence[0, "currentStep"].%X10 )
      Coil( "DB_Outputs".activeOutputsReq[10] )
   END_RUNG
   RUNG wire#powerrail
      Contact( "DB_Outputs".outputSequence[0, "currentStep"].%X11 )
      Coil( "DB_Outputs".activeOutputsReq[11] )
   END_RUNG
   RUNG wire#powerrail
      Contact( "DB_Outputs".outputSequence[0, "currentStep"].%X12 )
      Coil( "DB_Outputs".activeOutputsReq[12] )
   END_RUNG
   RUNG wire#powerrail
      Contact( "DB_Outputs".outputSequence[0, "currentStep"].%X13 )
      Coil( "DB_Outputs".activeOutputsReq[13] )
   END_RUNG
   RUNG wire#powerrail
      Contact( "DB_Outputs".outputSequence[0, "currentStep"].%X14 )
      Coil( "DB_Outputs".activeOutputsReq[14] )
   END_RUNG
   RUNG wire#powerrail
      Contact( "DB_Outputs".outputSequence[0, "currentStep"].%X15 )
      Coil( "DB_Outputs".activeOutputsReq[15] )
   END_RUNG
   RUNG wire#powerrail
      Contact( "DB_Outputs".outputSequence[0, "currentStep"].%X16 )
      Coil( "DB_Outputs".activeOutputsReq[16] )
   END_RUNG
   RUNG wire#powerrail
      Contact( "DB_Outputs".outputSequence[0, "currentStep"].%X17 )
      Coil( "DB_Outputs".activeOutputsReq[17] )
   END_RUNG
   RUNG wire#powerrail
      Contact( "DB_Outputs".outputSequence[0, "currentStep"].%X18 )
      Coil( "DB_Outputs".activeOutputsReq[18] )
   END_RUNG
   RUNG wire#powerrail
      Contact( "DB_Outputs".outputSequence[0, "currentStep"].%X19 )
      Coil( "DB_Outputs".activeOutputsReq[19] )
   END_RUNG
   RUNG wire#powerrail
      Contact( "DB_Outputs".outputSequence[0, "currentStep"].%X20 )
      Coil( "DB_Outputs".activeOutputsReq[20] )
   END_RUNG
   RUNG wire#powerrail
      Contact( "DB_Outputs".outputSequence[0, "currentStep"].%X21 )
      Coil( "DB_Outputs".activeOutputsReq[21] )
   END_RUNG
   RUNG wire#powerrail
      Contact( "DB_Outputs".outputSequence[0, "currentStep"].%X22 )
      Coil( "DB_Outputs".activeOutputsReq[22] )
   END_RUNG
   RUNG wire#powerrail
      Contact( "DB_Outputs".outputSequence[0, "currentStep"].%X23 )
      Coil( "DB_Outputs".activeOutputsReq[23] )
   END_RUNG
   RUNG wire#powerrail
      Contact( "DB_Outputs".outputSequence[0, "currentStep"].%X24 )
      Coil( "DB_Outputs".activeOutputsReq[24] )
   END_RUNG
   RUNG wire#powerrail
      Contact( "DB_Outputs".outputSequence[0, "currentStep"].%X25 )
      Coil( "DB_Outputs".activeOutputsReq[25] )
   END_RUNG
   RUNG wire#powerrail
      Contact( "DB_Outputs".outputSequence[0, "currentStep"].%X26 )
      Coil( "DB_Outputs".activeOutputsReq[26] )
   END_RUNG
   RUNG wire#powerrail
      Contact( "DB_Outputs".outputSequence[0, "currentStep"].%X27 )
      Coil( "DB_Outputs".activeOutputsReq[27] )
   END_RUNG
   RUNG wire#powerrail
      Contact( "DB_Outputs".outputSequence[0, "currentStep"].%X28 )
      Coil( "DB_Outputs".activeOutputsReq[28] )
   END_RUNG
   RUNG wire#powerrail
      Contact( "DB_Outputs".outputSequence[0, "currentStep"].%X29 )
      Coil( "DB_Outputs".activeOutputsReq[29] )
   END_RUNG
   RUNG wire#powerrail
      Contact( "DB_Outputs".outputSequence[0, "currentStep"].%X30 )
      Coil( "DB_Outputs".activeOutputsReq[30] )
   END_RUNG
   RUNG wire#powerrail
      Contact( "DB_Outputs".outputSequence[0, "currentStep"].%X31 )
      Coil( "DB_Outputs".activeOutputsReq[31] )
   END_RUNG
   // the same network as SCL:
   "DB_Outputs".activeOutputsReq[0] := "DB_Outputs".outputSequence[0, "currentStep"].%X0;
   "DB_Outputs".activeOutputsReq[1] := "DB_Outputs".outputSequence[0, "currentStep"].%X1;
   "DB_Outputs".activeOutputsReq[2] := "DB_Outputs".outputSequence[0, "currentStep"].%X2;
   "DB_Outputs".activeOutputsReq[3] := "DB_Outputs".outputSequence[0, "currentStep"].%X3;
   "DB_Outputs".activeOutputsReq[4] := "DB_Outputs".outputSequence[0, "currentStep"].%X4;
   "DB_Outputs".activeOutputsReq[5] := "DB_Outputs".outputSequence[0, "currentStep"].%X5;
   "DB_Outputs".activeOutputsReq[6] := "DB_Outputs".outputSequence[0, "currentStep"].%X6;
   "DB_Outputs".activeOutputsReq[7] := "DB_Outputs".outputSequence[0, "currentStep"].%X7;
   "DB_Outputs".activeOutputsReq[8] := "DB_Outputs".outputSequence[0, "currentStep"].%X8;
   "DB_Outputs".activeOutputsReq[9] := "DB_Outputs".outputSequence[0, "currentStep"].%X9;
   "DB_Outputs".activeOutputsReq[10] := "DB_Outputs".outputSequence[0, "currentStep"].%X10;
   "DB_Outputs".activeOutputsReq[11] := "DB_Outputs".outputSequence[0, "currentStep"].%X11;
   "DB_Outputs".activeOutputsReq[12] := "DB_Outputs".outputSequence[0, "currentStep"].%X12;
   "DB_Outputs".activeOutputsReq[13] := "DB_Outputs".outputSequence[0, "currentStep"].%X13;
   "DB_Outputs".activeOutputsReq[14] := "DB_Outputs".outputSequence[0, "currentStep"].%X14;
   "DB_Outputs".activeOutputsReq[15] := "DB_Outputs".outputSequence[0, "currentStep"].%X15;
   "DB_Outputs".activeOutputsReq[16] := "DB_Outputs".outputSequence[0, "currentStep"].%X16;
   "DB_Outputs".activeOutputsReq[17] := "DB_Outputs".outputSequence[0, "currentStep"].%X17;
   "DB_Outputs".activeOutputsReq[18] := "DB_Outputs".outputSequence[0, "currentStep"].%X18;
   "DB_Outputs".activeOutputsReq[19] := "DB_Outputs".outputSequence[0, "currentStep"].%X19;
   "DB_Outputs".activeOutputsReq[20] := "DB_Outputs".outputSequence[0, "currentStep"].%X20;
   "DB_Outputs".activeOutputsReq[21] := "DB_Outputs".outputSequence[0, "currentStep"].%X21;
   "DB_Outputs".activeOutputsReq[22] := "DB_Outputs".outputSequence[0, "currentStep"].%X22;
   "DB_Outputs".activeOutputsReq[23] := "DB_Outputs".outputSequence[0, "currentStep"].%X23;
   "DB_Outputs".activeOutputsReq[24] := "DB_Outputs".outputSequence[0, "currentStep"].%X24;
   "DB_Outputs".activeOutputsReq[25] := "DB_Outputs".outputSequence[0, "currentStep"].%X25;
   "DB_Outputs".activeOutputsReq[26] := "DB_Outputs".outputSequence[0, "currentStep"].%X26;
   "DB_Outputs".activeOutputsReq[27] := "DB_Outputs".outputSequence[0, "currentStep"].%X27;
   "DB_Outputs".activeOutputsReq[28] := "DB_Outputs".outputSequence[0, "currentStep"].%X28;
   "DB_Outputs".activeOutputsReq[29] := "DB_Outputs".outputSequence[0, "currentStep"].%X29;
   "DB_Outputs".activeOutputsReq[30] := "DB_Outputs".outputSequence[0, "currentStep"].%X30;
   "DB_Outputs".activeOutputsReq[31] := "DB_Outputs".outputSequence[0, "currentStep"].%X31;
END_REGION

REGION Network 4: MASK OUTPUTS STATUS
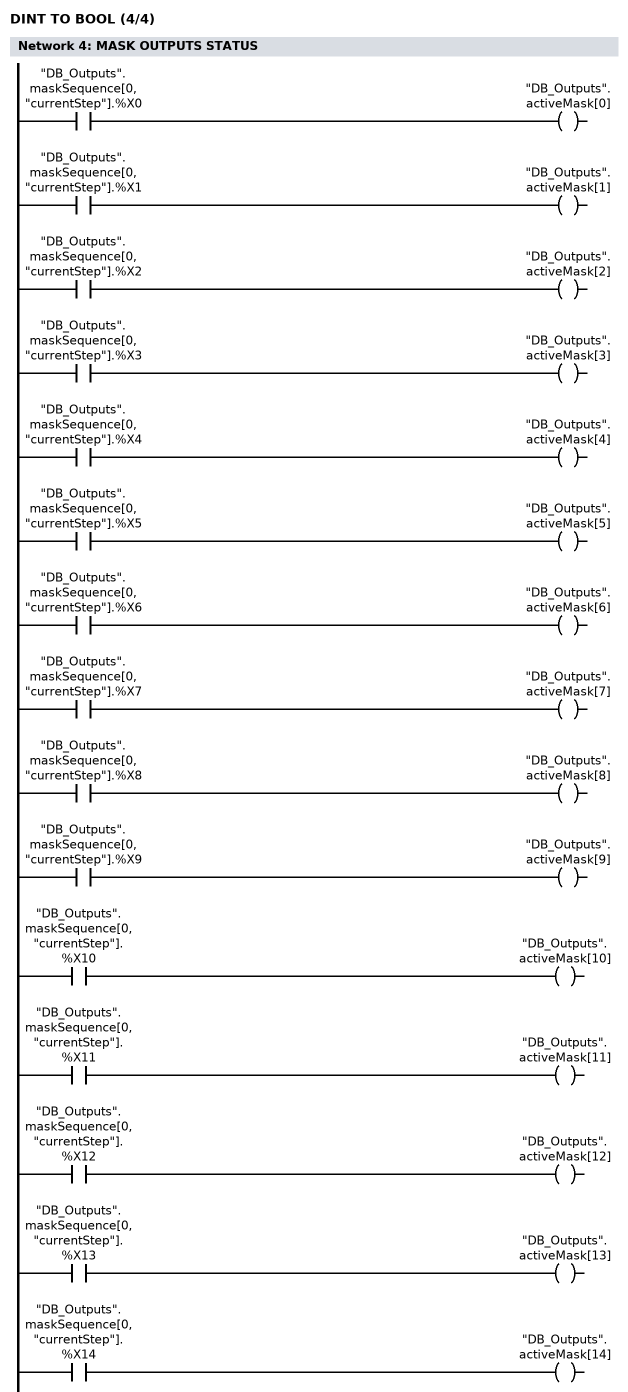
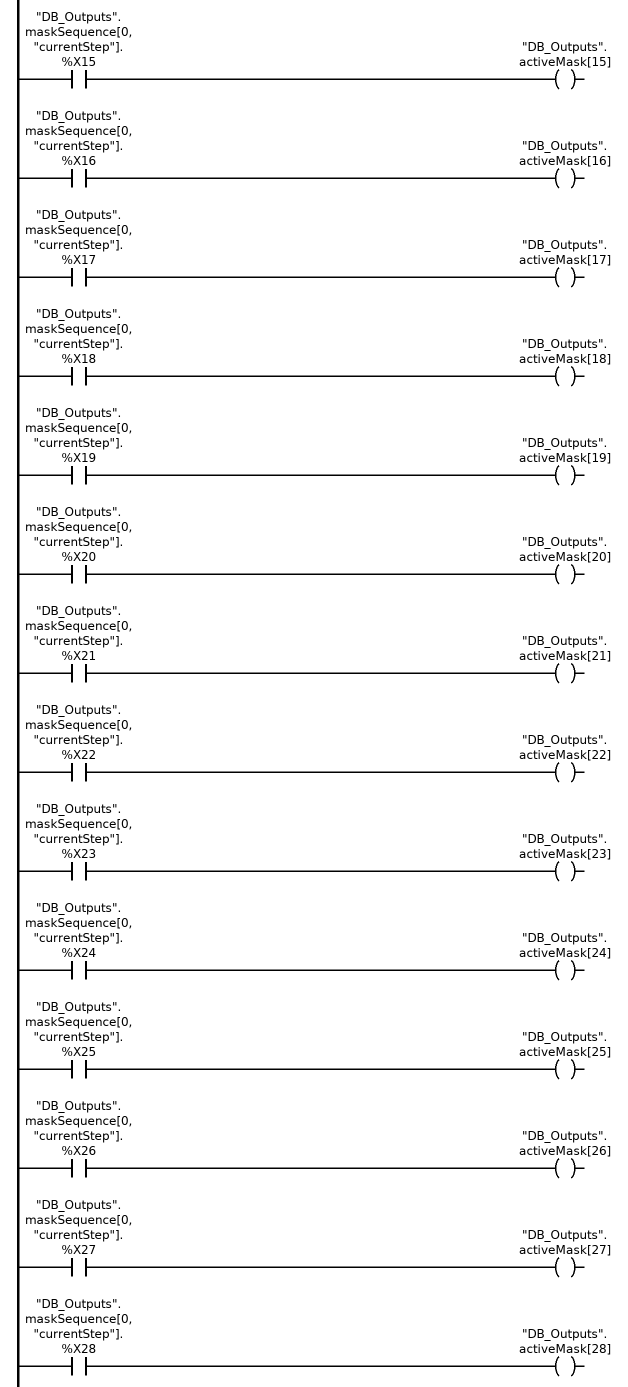
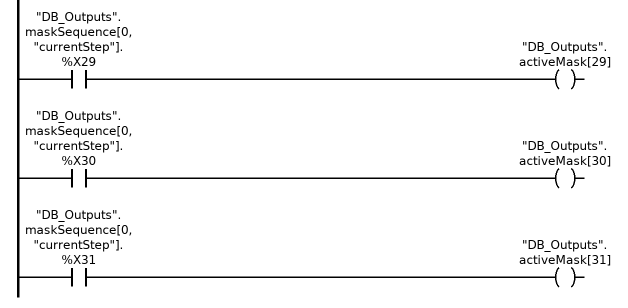
   RUNG wire#powerrail
      Contact( "DB_Outputs".maskSequence[0, "currentStep"].%X0 )
      Coil( "DB_Outputs".activeMask[0] )
   END_RUNG
   RUNG wire#powerrail
      Contact( "DB_Outputs".maskSequence[0, "currentStep"].%X1 )
      Coil( "DB_Outputs".activeMask[1] )
   END_RUNG
   RUNG wire#powerrail
      Contact( "DB_Outputs".maskSequence[0, "currentStep"].%X2 )
      Coil( "DB_Outputs".activeMask[2] )
   END_RUNG
   RUNG wire#powerrail
      Contact( "DB_Outputs".maskSequence[0, "currentStep"].%X3 )
      Coil( "DB_Outputs".activeMask[3] )
   END_RUNG
   RUNG wire#powerrail
      Contact( "DB_Outputs".maskSequence[0, "currentStep"].%X4 )
      Coil( "DB_Outputs".activeMask[4] )
   END_RUNG
   RUNG wire#powerrail
      Contact( "DB_Outputs".maskSequence[0, "currentStep"].%X5 )
      Coil( "DB_Outputs".activeMask[5] )
   END_RUNG
   RUNG wire#powerrail
      Contact( "DB_Outputs".maskSequence[0, "currentStep"].%X6 )
      Coil( "DB_Outputs".activeMask[6] )
   END_RUNG
   RUNG wire#powerrail
      Contact( "DB_Outputs".maskSequence[0, "currentStep"].%X7 )
      Coil( "DB_Outputs".activeMask[7] )
   END_RUNG
   RUNG wire#powerrail
      Contact( "DB_Outputs".maskSequence[0, "currentStep"].%X8 )
      Coil( "DB_Outputs".activeMask[8] )
   END_RUNG
   RUNG wire#powerrail
      Contact( "DB_Outputs".maskSequence[0, "currentStep"].%X9 )
      Coil( "DB_Outputs".activeMask[9] )
   END_RUNG
   RUNG wire#powerrail
      Contact( "DB_Outputs".maskSequence[0, "currentStep"].%X10 )
      Coil( "DB_Outputs".activeMask[10] )
   END_RUNG
   RUNG wire#powerrail
      Contact( "DB_Outputs".maskSequence[0, "currentStep"].%X11 )
      Coil( "DB_Outputs".activeMask[11] )
   END_RUNG
   RUNG wire#powerrail
      Contact( "DB_Outputs".maskSequence[0, "currentStep"].%X12 )
      Coil( "DB_Outputs".activeMask[12] )
   END_RUNG
   RUNG wire#powerrail
      Contact( "DB_Outputs".maskSequence[0, "currentStep"].%X13 )
      Coil( "DB_Outputs".activeMask[13] )
   END_RUNG
   RUNG wire#powerrail
      Contact( "DB_Outputs".maskSequence[0, "currentStep"].%X14 )
      Coil( "DB_Outputs".activeMask[14] )
   END_RUNG
   RUNG wire#powerrail
      Contact( "DB_Outputs".maskSequence[0, "currentStep"].%X15 )
      Coil( "DB_Outputs".activeMask[15] )
   END_RUNG
   RUNG wire#powerrail
      Contact( "DB_Outputs".maskSequence[0, "currentStep"].%X16 )
      Coil( "DB_Outputs".activeMask[16] )
   END_RUNG
   RUNG wire#powerrail
      Contact( "DB_Outputs".maskSequence[0, "currentStep"].%X17 )
      Coil( "DB_Outputs".activeMask[17] )
   END_RUNG
   RUNG wire#powerrail
      Contact( "DB_Outputs".maskSequence[0, "currentStep"].%X18 )
      Coil( "DB_Outputs".activeMask[18] )
   END_RUNG
   RUNG wire#powerrail
      Contact( "DB_Outputs".maskSequence[0, "currentStep"].%X19 )
      Coil( "DB_Outputs".activeMask[19] )
   END_RUNG
   RUNG wire#powerrail
      Contact( "DB_Outputs".maskSequence[0, "currentStep"].%X20 )
      Coil( "DB_Outputs".activeMask[20] )
   END_RUNG
   RUNG wire#powerrail
      Contact( "DB_Outputs".maskSequence[0, "currentStep"].%X21 )
      Coil( "DB_Outputs".activeMask[21] )
   END_RUNG
   RUNG wire#powerrail
      Contact( "DB_Outputs".maskSequence[0, "currentStep"].%X22 )
      Coil( "DB_Outputs".activeMask[22] )
   END_RUNG
   RUNG wire#powerrail
      Contact( "DB_Outputs".maskSequence[0, "currentStep"].%X23 )
      Coil( "DB_Outputs".activeMask[23] )
   END_RUNG
   RUNG wire#powerrail
      Contact( "DB_Outputs".maskSequence[0, "currentStep"].%X24 )
      Coil( "DB_Outputs".activeMask[24] )
   END_RUNG
   RUNG wire#powerrail
      Contact( "DB_Outputs".maskSequence[0, "currentStep"].%X25 )
      Coil( "DB_Outputs".activeMask[25] )
   END_RUNG
   RUNG wire#powerrail
      Contact( "DB_Outputs".maskSequence[0, "currentStep"].%X26 )
      Coil( "DB_Outputs".activeMask[26] )
   END_RUNG
   RUNG wire#powerrail
      Contact( "DB_Outputs".maskSequence[0, "currentStep"].%X27 )
      Coil( "DB_Outputs".activeMask[27] )
   END_RUNG
   RUNG wire#powerrail
      Contact( "DB_Outputs".maskSequence[0, "currentStep"].%X28 )
      Coil( "DB_Outputs".activeMask[28] )
   END_RUNG
   RUNG wire#powerrail
      Contact( "DB_Outputs".maskSequence[0, "currentStep"].%X29 )
      Coil( "DB_Outputs".activeMask[29] )
   END_RUNG
   RUNG wire#powerrail
      Contact( "DB_Outputs".maskSequence[0, "currentStep"].%X30 )
      Coil( "DB_Outputs".activeMask[30] )
   END_RUNG
   RUNG wire#powerrail
      Contact( "DB_Outputs".maskSequence[0, "currentStep"].%X31 )
      Coil( "DB_Outputs".activeMask[31] )
   END_RUNG
   // the same network as SCL:
   "DB_Outputs".activeMask[0] := "DB_Outputs".maskSequence[0, "currentStep"].%X0;
   "DB_Outputs".activeMask[1] := "DB_Outputs".maskSequence[0, "currentStep"].%X1;
   "DB_Outputs".activeMask[2] := "DB_Outputs".maskSequence[0, "currentStep"].%X2;
   "DB_Outputs".activeMask[3] := "DB_Outputs".maskSequence[0, "currentStep"].%X3;
   "DB_Outputs".activeMask[4] := "DB_Outputs".maskSequence[0, "currentStep"].%X4;
   "DB_Outputs".activeMask[5] := "DB_Outputs".maskSequence[0, "currentStep"].%X5;
   "DB_Outputs".activeMask[6] := "DB_Outputs".maskSequence[0, "currentStep"].%X6;
   "DB_Outputs".activeMask[7] := "DB_Outputs".maskSequence[0, "currentStep"].%X7;
   "DB_Outputs".activeMask[8] := "DB_Outputs".maskSequence[0, "currentStep"].%X8;
   "DB_Outputs".activeMask[9] := "DB_Outputs".maskSequence[0, "currentStep"].%X9;
   "DB_Outputs".activeMask[10] := "DB_Outputs".maskSequence[0, "currentStep"].%X10;
   "DB_Outputs".activeMask[11] := "DB_Outputs".maskSequence[0, "currentStep"].%X11;
   "DB_Outputs".activeMask[12] := "DB_Outputs".maskSequence[0, "currentStep"].%X12;
   "DB_Outputs".activeMask[13] := "DB_Outputs".maskSequence[0, "currentStep"].%X13;
   "DB_Outputs".activeMask[14] := "DB_Outputs".maskSequence[0, "currentStep"].%X14;
   "DB_Outputs".activeMask[15] := "DB_Outputs".maskSequence[0, "currentStep"].%X15;
   "DB_Outputs".activeMask[16] := "DB_Outputs".maskSequence[0, "currentStep"].%X16;
   "DB_Outputs".activeMask[17] := "DB_Outputs".maskSequence[0, "currentStep"].%X17;
   "DB_Outputs".activeMask[18] := "DB_Outputs".maskSequence[0, "currentStep"].%X18;
   "DB_Outputs".activeMask[19] := "DB_Outputs".maskSequence[0, "currentStep"].%X19;
   "DB_Outputs".activeMask[20] := "DB_Outputs".maskSequence[0, "currentStep"].%X20;
   "DB_Outputs".activeMask[21] := "DB_Outputs".maskSequence[0, "currentStep"].%X21;
   "DB_Outputs".activeMask[22] := "DB_Outputs".maskSequence[0, "currentStep"].%X22;
   "DB_Outputs".activeMask[23] := "DB_Outputs".maskSequence[0, "currentStep"].%X23;
   "DB_Outputs".activeMask[24] := "DB_Outputs".maskSequence[0, "currentStep"].%X24;
   "DB_Outputs".activeMask[25] := "DB_Outputs".maskSequence[0, "currentStep"].%X25;
   "DB_Outputs".activeMask[26] := "DB_Outputs".maskSequence[0, "currentStep"].%X26;
   "DB_Outputs".activeMask[27] := "DB_Outputs".maskSequence[0, "currentStep"].%X27;
   "DB_Outputs".activeMask[28] := "DB_Outputs".maskSequence[0, "currentStep"].%X28;
   "DB_Outputs".activeMask[29] := "DB_Outputs".maskSequence[0, "currentStep"].%X29;
   "DB_Outputs".activeMask[30] := "DB_Outputs".maskSequence[0, "currentStep"].%X30;
   "DB_Outputs".activeMask[31] := "DB_Outputs".maskSequence[0, "currentStep"].%X31;
END_REGION
END_FUNCTION

FUNCTION "stationAlarms" : Void   // FC2, LAD
{ S7_Optimized_Access := 'TRUE' }
VERSION : 0.1
// stored: AutoNumber true, IsIECCheckEnabled false, SetENOAutomatically false, UDAEnableTagReadback false
   VAR_TEMP   // added for the SCL form of the ladder/FBD networks
      _w1 : Bool;
      _w2 : Bool;
      _w3 : Bool;
      _w4 : Bool;
      _w5 : Bool;
   END_VAR
BEGIN

REGION Network 1: ACTIVE ALARM
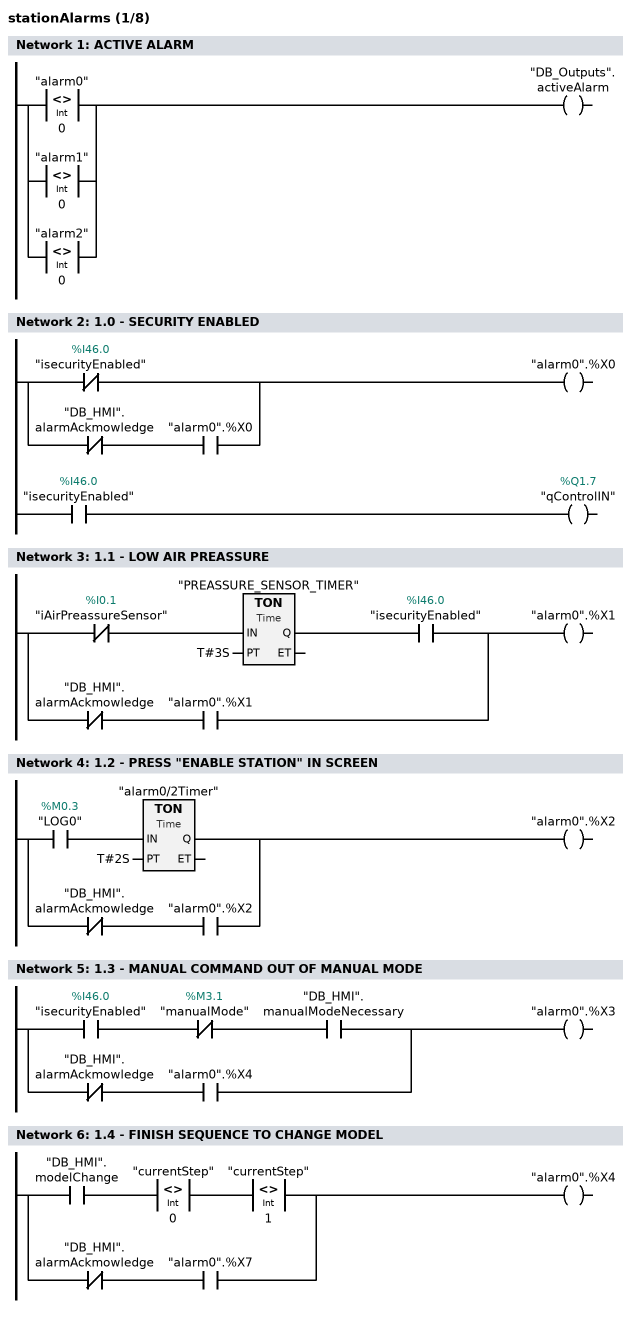
   RUNG wire#powerrail
      { S7_Templates := "SrcType := Int" } NE_Contact(in1 := "alarm0", in2 := 0)
      wire#w1
      Coil( "DB_Outputs".activeAlarm )
   END_RUNG
   RUNG wire#powerrail
      { S7_Templates := "SrcType := Int" } NE_Contact(in1 := "alarm1", in2 := 0)
   END_RUNG wire#w1
   RUNG wire#powerrail
      { S7_Templates := "SrcType := Int" } NE_Contact(in1 := "alarm2", in2 := 0)
   END_RUNG wire#w1
   // the same network as SCL:
   "DB_Outputs".activeAlarm := ("alarm0" <> 0) OR ("alarm1" <> 0) OR ("alarm2" <> 0);
END_REGION

REGION Network 2: 1.0 - SECURITY ENABLED
   RUNG wire#powerrail
      I_Contact( "isecurityEnabled" )
      wire#w1
      Coil( "alarm0".%X0 )
   END_RUNG
   RUNG wire#powerrail
      I_Contact( "DB_HMI".alarmAckmowledge )
      Contact( "alarm0".%X0 )
   END_RUNG wire#w1
   RUNG wire#powerrail
      Contact( "isecurityEnabled" )
      Coil( "qControlIN" )
   END_RUNG
   // the same network as SCL:
   "alarm0".%X0 := NOT "isecurityEnabled" OR (NOT "DB_HMI".alarmAckmowledge AND "alarm0".%X0);
   "qControlIN" := "isecurityEnabled";
END_REGION

REGION Network 3: 1.1 - LOW AIR PREASSURE
   RUNG wire#powerrail
      I_Contact( "iAirPreassureSensor" )
      { S7_Templates := "time_type := Time" } "PREASSURE_SENSOR_TIMER".TON(pt := T#3S, et =>)
      Contact( "isecurityEnabled" )
      wire#w1
      Coil( "alarm0".%X1 )
   END_RUNG
   RUNG wire#powerrail
      I_Contact( "DB_HMI".alarmAckmowledge )
      Contact( "alarm0".%X1 )
   END_RUNG wire#w1
   // the same network as SCL:
   "PREASSURE_SENSOR_TIMER".TON(IN := NOT "iAirPreassureSensor", PT := T#3S);
   "alarm0".%X1 := ("PREASSURE_SENSOR_TIMER".Q AND "isecurityEnabled") OR (NOT "DB_HMI".alarmAckmowledge AND "alarm0".%X1);
END_REGION

REGION Network 4: 1.2 - PRESS "ENABLE STATION" IN SCREEN
   RUNG wire#powerrail
      Contact( "LOG0" )
      { S7_Templates := "time_type := Time" } "alarm0/2Timer".TON(pt := T#2S, et =>)
      wire#w1
      Coil( "alarm0".%X2 )
   END_RUNG
   RUNG wire#powerrail
      I_Contact( "DB_HMI".alarmAckmowledge )
      Contact( "alarm0".%X2 )
   END_RUNG wire#w1
   // the same network as SCL:
   "alarm0/2Timer".TON(IN := "LOG0", PT := T#2S);
   "alarm0".%X2 := "alarm0/2Timer".Q OR (NOT "DB_HMI".alarmAckmowledge AND "alarm0".%X2);
END_REGION

REGION Network 5: 1.3 - MANUAL COMMAND OUT OF MANUAL MODE
   RUNG wire#powerrail
      Contact( "isecurityEnabled" )
      I_Contact( "manualMode" )
      Contact( "DB_HMI".manualModeNecessary )
      wire#w1
      Coil( "alarm0".%X3 )
   END_RUNG
   RUNG wire#powerrail
      I_Contact( "DB_HMI".alarmAckmowledge )
      Contact( "alarm0".%X4 )
   END_RUNG wire#w1
   // the same network as SCL:
   "alarm0".%X3 := ("isecurityEnabled" AND NOT "manualMode" AND "DB_HMI".manualModeNecessary) OR (NOT "DB_HMI".alarmAckmowledge AND "alarm0".%X4);
END_REGION

REGION Network 6: 1.4 - FINISH SEQUENCE TO CHANGE MODEL
   RUNG wire#powerrail
      Contact( "DB_HMI".modelChange )
      { S7_Templates := "SrcType := Int" } NE_Contact(in1 := "currentStep", in2 := 0)
      { S7_Templates := "SrcType := Int" } NE_Contact(in1 := "currentStep", in2 := 1)
      wire#w1
      Coil( "alarm0".%X4 )
   END_RUNG
   RUNG wire#powerrail
      I_Contact( "DB_HMI".alarmAckmowledge )
      Contact( "alarm0".%X7 )
   END_RUNG wire#w1
   // the same network as SCL:
   "alarm0".%X4 := ("DB_HMI".modelChange AND ("currentStep" <> 0) AND ("currentStep" <> 1)) OR (NOT "DB_HMI".alarmAckmowledge AND "alarm0".%X7);
END_REGION

REGION Network 7: 1.5 - WRONG LABEL
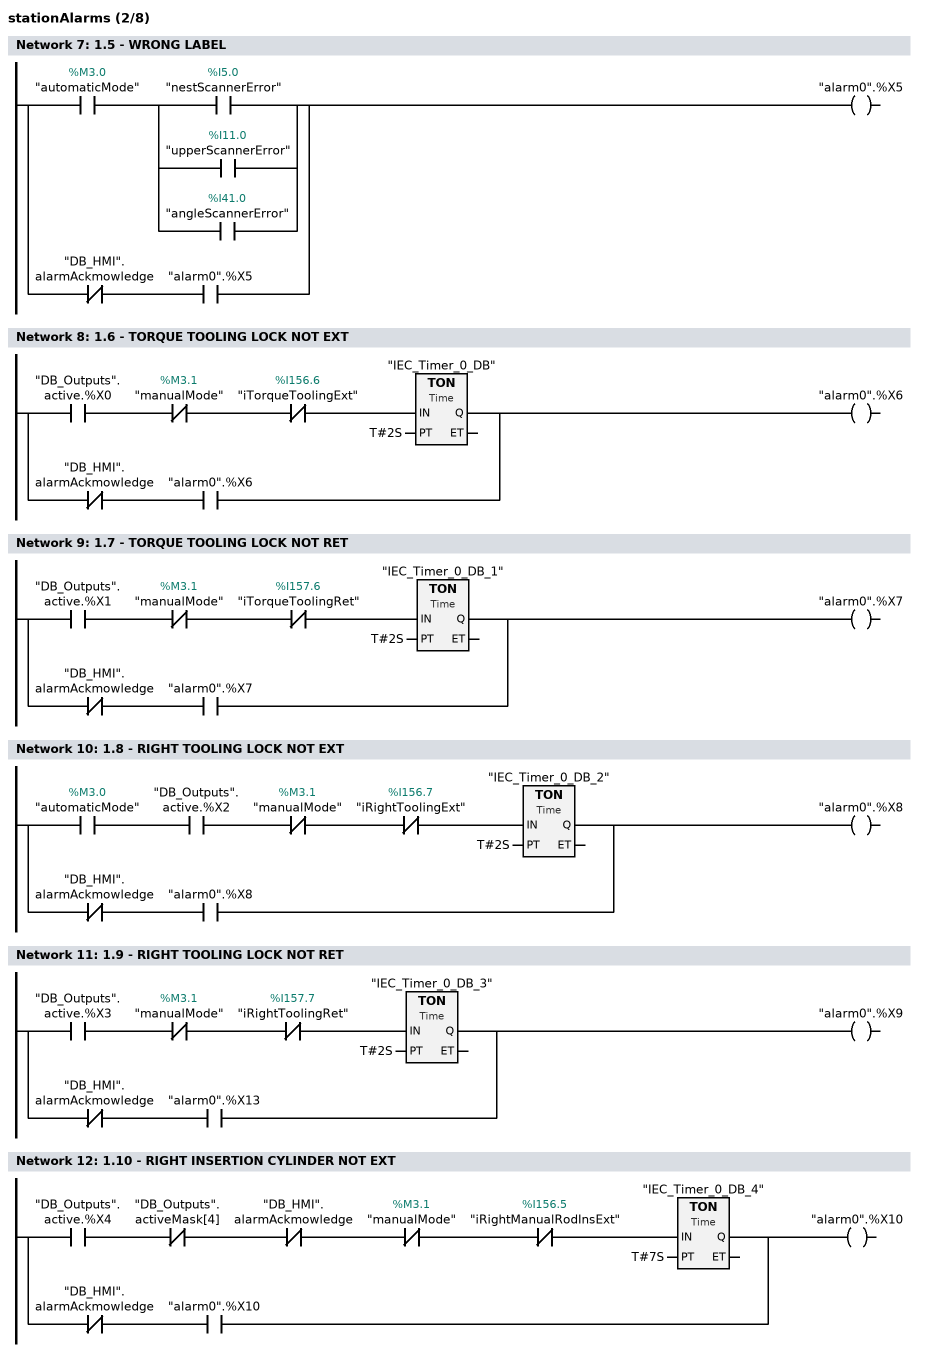
   RUNG wire#powerrail
      Contact( "automaticMode" )
      wire#w1
      Contact( "nestScannerError" )
      wire#w2
      Coil( "alarm0".%X5 )
   END_RUNG
   RUNG wire#w1
      Contact( "upperScannerError" )
   END_RUNG wire#w2
   RUNG wire#w1
      Contact( "angleScannerError" )
   END_RUNG wire#w2
   RUNG wire#powerrail
      I_Contact( "DB_HMI".alarmAckmowledge )
      Contact( "alarm0".%X5 )
   END_RUNG wire#w2
   // the same network as SCL:
   "alarm0".%X5 := ("automaticMode" AND ("nestScannerError" OR "upperScannerError" OR "angleScannerError")) OR (NOT "DB_HMI".alarmAckmowledge AND "alarm0".%X5);
END_REGION

REGION Network 8: 1.6 - TORQUE TOOLING LOCK NOT EXT
   RUNG wire#powerrail
      Contact( "DB_Outputs".active.%X0 )
      I_Contact( "manualMode" )
      I_Contact( "iTorqueToolingExt" )
      { S7_Templates := "time_type := Time" } "IEC_Timer_0_DB".TON(pt := T#2S, et =>)
      wire#w1
      Coil( "alarm0".%X6 )
   END_RUNG
   RUNG wire#powerrail
      I_Contact( "DB_HMI".alarmAckmowledge )
      Contact( "alarm0".%X6 )
   END_RUNG wire#w1
   // the same network as SCL:
   "IEC_Timer_0_DB".TON(IN := "DB_Outputs".active.%X0 AND NOT "manualMode" AND NOT "iTorqueToolingExt",
                        PT := T#2S);
   "alarm0".%X6 := "IEC_Timer_0_DB".Q OR (NOT "DB_HMI".alarmAckmowledge AND "alarm0".%X6);
END_REGION

REGION Network 9: 1.7 - TORQUE TOOLING LOCK NOT RET
   RUNG wire#powerrail
      Contact( "DB_Outputs".active.%X1 )
      I_Contact( "manualMode" )
      I_Contact( "iTorqueToolingRet" )
      { S7_Templates := "time_type := Time" } "IEC_Timer_0_DB_1".TON(pt := T#2S, et =>)
      wire#w1
      Coil( "alarm0".%X7 )
   END_RUNG
   RUNG wire#powerrail
      I_Contact( "DB_HMI".alarmAckmowledge )
      Contact( "alarm0".%X7 )
   END_RUNG wire#w1
   // the same network as SCL:
   "IEC_Timer_0_DB_1".TON(IN := "DB_Outputs".active.%X1 AND NOT "manualMode" AND NOT "iTorqueToolingRet",
                          PT := T#2S);
   "alarm0".%X7 := "IEC_Timer_0_DB_1".Q OR (NOT "DB_HMI".alarmAckmowledge AND "alarm0".%X7);
END_REGION

REGION Network 10: 1.8 - RIGHT TOOLING LOCK NOT EXT
   RUNG wire#powerrail
      Contact( "automaticMode" )
      Contact( "DB_Outputs".active.%X2 )
      I_Contact( "manualMode" )
      I_Contact( "iRightToolingExt" )
      { S7_Templates := "time_type := Time" } "IEC_Timer_0_DB_2".TON(pt := T#2S, et =>)
      wire#w1
      Coil( "alarm0".%X8 )
   END_RUNG
   RUNG wire#powerrail
      I_Contact( "DB_HMI".alarmAckmowledge )
      Contact( "alarm0".%X8 )
   END_RUNG wire#w1
   // the same network as SCL:
   "IEC_Timer_0_DB_2".TON(IN := "automaticMode" AND "DB_Outputs".active.%X2 AND NOT "manualMode" AND NOT "iRightToolingExt",
                          PT := T#2S);
   "alarm0".%X8 := "IEC_Timer_0_DB_2".Q OR (NOT "DB_HMI".alarmAckmowledge AND "alarm0".%X8);
END_REGION

REGION Network 11: 1.9 - RIGHT TOOLING LOCK NOT RET
   RUNG wire#powerrail
      Contact( "DB_Outputs".active.%X3 )
      I_Contact( "manualMode" )
      I_Contact( "iRightToolingRet" )
      { S7_Templates := "time_type := Time" } "IEC_Timer_0_DB_3".TON(pt := T#2S, et =>)
      wire#w1
      Coil( "alarm0".%X9 )
   END_RUNG
   RUNG wire#powerrail
      I_Contact( "DB_HMI".alarmAckmowledge )
      Contact( "alarm0".%X13 )
   END_RUNG wire#w1
   // the same network as SCL:
   "IEC_Timer_0_DB_3".TON(IN := "DB_Outputs".active.%X3 AND NOT "manualMode" AND NOT "iRightToolingRet",
                          PT := T#2S);
   "alarm0".%X9 := "IEC_Timer_0_DB_3".Q OR (NOT "DB_HMI".alarmAckmowledge AND "alarm0".%X13);
END_REGION

REGION Network 12: 1.10 - RIGHT INSERTION CYLINDER NOT EXT
   RUNG wire#powerrail
      Contact( "DB_Outputs".active.%X4 )
      I_Contact( "DB_Outputs".activeMask[4] )
      I_Contact( "DB_HMI".alarmAckmowledge )
      I_Contact( "manualMode" )
      I_Contact( "iRightManualRodInsExt" )
      { S7_Templates := "time_type := Time" } "IEC_Timer_0_DB_4".TON(pt := T#7S, et =>)
      wire#w1
      Coil( "alarm0".%X10 )
   END_RUNG
   RUNG wire#powerrail
      I_Contact( "DB_HMI".alarmAckmowledge )
      Contact( "alarm0".%X10 )
   END_RUNG wire#w1
   // the same network as SCL:
   "IEC_Timer_0_DB_4".TON(IN := "DB_Outputs".active.%X4 AND NOT "DB_Outputs".activeMask[4] AND NOT "DB_HMI".alarmAckmowledge AND NOT "manualMode" AND NOT "iRightManualRodInsExt",
                          PT := T#7S);
   "alarm0".%X10 := "IEC_Timer_0_DB_4".Q OR (NOT "DB_HMI".alarmAckmowledge AND "alarm0".%X10);
END_REGION

REGION Network 13: 1.11 - RIGHT INSERTION CYLINDER NOT RET
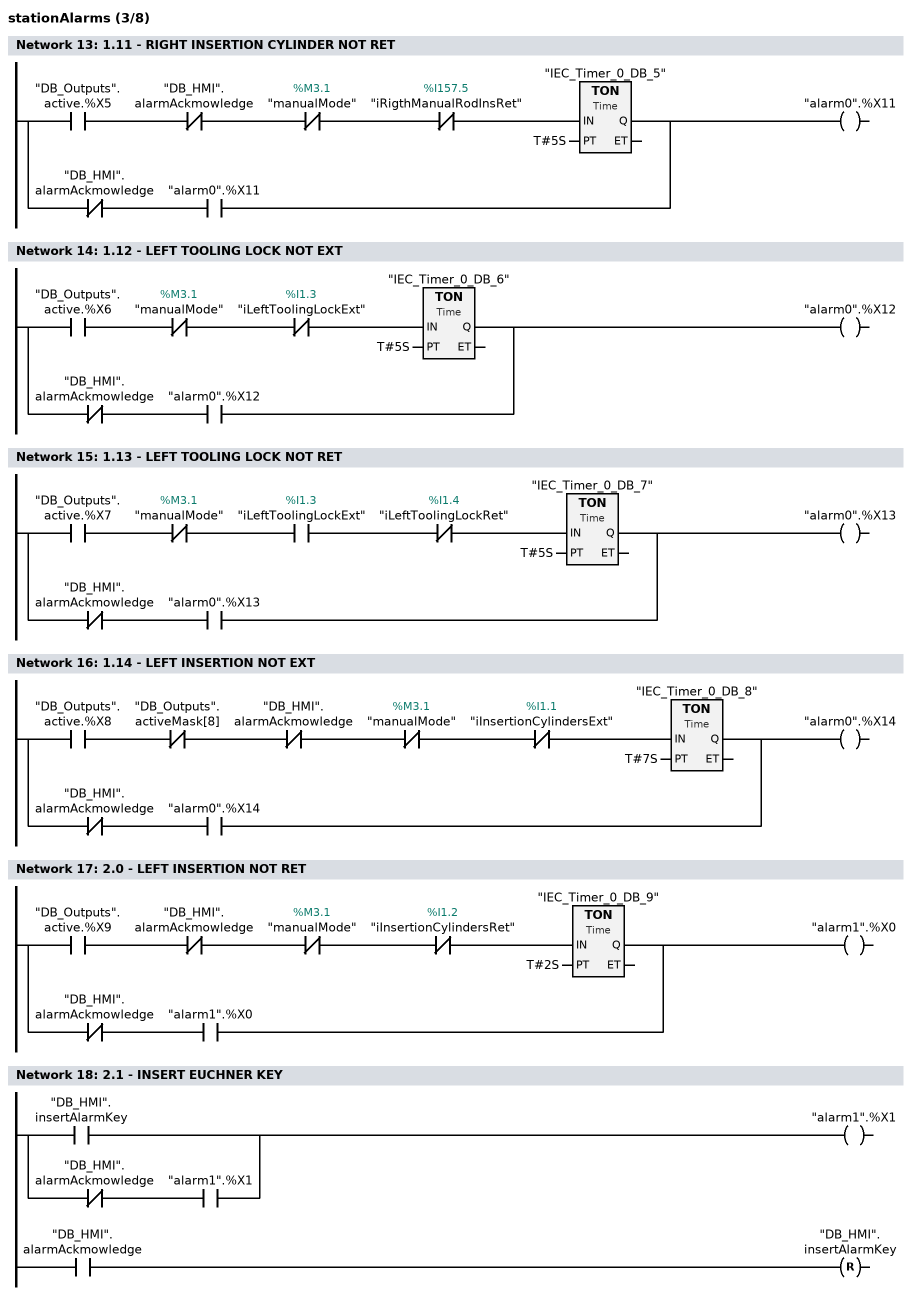
   RUNG wire#powerrail
      Contact( "DB_Outputs".active.%X5 )
      I_Contact( "DB_HMI".alarmAckmowledge )
      I_Contact( "manualMode" )
      I_Contact( "iRigthManualRodInsRet" )
      { S7_Templates := "time_type := Time" } "IEC_Timer_0_DB_5".TON(pt := T#5S, et =>)
      wire#w1
      Coil( "alarm0".%X11 )
   END_RUNG
   RUNG wire#powerrail
      I_Contact( "DB_HMI".alarmAckmowledge )
      Contact( "alarm0".%X11 )
   END_RUNG wire#w1
   // the same network as SCL:
   "IEC_Timer_0_DB_5".TON(IN := "DB_Outputs".active.%X5 AND NOT "DB_HMI".alarmAckmowledge AND NOT "manualMode" AND NOT "iRigthManualRodInsRet",
                          PT := T#5S);
   "alarm0".%X11 := "IEC_Timer_0_DB_5".Q OR (NOT "DB_HMI".alarmAckmowledge AND "alarm0".%X11);
END_REGION

REGION Network 14: 1.12 - LEFT TOOLING LOCK NOT EXT
   RUNG wire#powerrail
      Contact( "DB_Outputs".active.%X6 )
      I_Contact( "manualMode" )
      I_Contact( "iLeftToolingLockExt" )
      { S7_Templates := "time_type := Time" } "IEC_Timer_0_DB_6".TON(pt := T#5S, et =>)
      wire#w1
      Coil( "alarm0".%X12 )
   END_RUNG
   RUNG wire#powerrail
      I_Contact( "DB_HMI".alarmAckmowledge )
      Contact( "alarm0".%X12 )
   END_RUNG wire#w1
   // the same network as SCL:
   "IEC_Timer_0_DB_6".TON(IN := "DB_Outputs".active.%X6 AND NOT "manualMode" AND NOT "iLeftToolingLockExt",
                          PT := T#5S);
   "alarm0".%X12 := "IEC_Timer_0_DB_6".Q OR (NOT "DB_HMI".alarmAckmowledge AND "alarm0".%X12);
END_REGION

REGION Network 15: 1.13 - LEFT TOOLING LOCK NOT RET
   RUNG wire#powerrail
      Contact( "DB_Outputs".active.%X7 )
      I_Contact( "manualMode" )
      Contact( "iLeftToolingLockExt" )
      I_Contact( "iLeftToolingLockRet" )
      { S7_Templates := "time_type := Time" } "IEC_Timer_0_DB_7".TON(pt := T#5S, et =>)
      wire#w1
      Coil( "alarm0".%X13 )
   END_RUNG
   RUNG wire#powerrail
      I_Contact( "DB_HMI".alarmAckmowledge )
      Contact( "alarm0".%X13 )
   END_RUNG wire#w1
   // the same network as SCL:
   "IEC_Timer_0_DB_7".TON(IN := "DB_Outputs".active.%X7 AND NOT "manualMode" AND "iLeftToolingLockExt" AND NOT "iLeftToolingLockRet",
                          PT := T#5S);
   "alarm0".%X13 := "IEC_Timer_0_DB_7".Q OR (NOT "DB_HMI".alarmAckmowledge AND "alarm0".%X13);
END_REGION

REGION Network 16: 1.14 - LEFT INSERTION NOT EXT
   RUNG wire#powerrail
      Contact( "DB_Outputs".active.%X8 )
      I_Contact( "DB_Outputs".activeMask[8] )
      I_Contact( "DB_HMI".alarmAckmowledge )
      I_Contact( "manualMode" )
      I_Contact( "iInsertionCylindersExt" )
      { S7_Templates := "time_type := Time" } "IEC_Timer_0_DB_8".TON(pt := T#7S, et =>)
      wire#w1
      Coil( "alarm0".%X14 )
   END_RUNG
   RUNG wire#powerrail
      I_Contact( "DB_HMI".alarmAckmowledge )
      Contact( "alarm0".%X14 )
   END_RUNG wire#w1
   // the same network as SCL:
   "IEC_Timer_0_DB_8".TON(IN := "DB_Outputs".active.%X8 AND NOT "DB_Outputs".activeMask[8] AND NOT "DB_HMI".alarmAckmowledge AND NOT "manualMode" AND NOT "iInsertionCylindersExt",
                          PT := T#7S);
   "alarm0".%X14 := "IEC_Timer_0_DB_8".Q OR (NOT "DB_HMI".alarmAckmowledge AND "alarm0".%X14);
END_REGION

REGION Network 17: 2.0 - LEFT INSERTION NOT RET
   RUNG wire#powerrail
      Contact( "DB_Outputs".active.%X9 )
      I_Contact( "DB_HMI".alarmAckmowledge )
      I_Contact( "manualMode" )
      I_Contact( "iInsertionCylindersRet" )
      { S7_Templates := "time_type := Time" } "IEC_Timer_0_DB_9".TON(pt := T#2S, et =>)
      wire#w1
      Coil( "alarm1".%X0 )
   END_RUNG
   RUNG wire#powerrail
      I_Contact( "DB_HMI".alarmAckmowledge )
      Contact( "alarm1".%X0 )
   END_RUNG wire#w1
   // the same network as SCL:
   "IEC_Timer_0_DB_9".TON(IN := "DB_Outputs".active.%X9 AND NOT "DB_HMI".alarmAckmowledge AND NOT "manualMode" AND NOT "iInsertionCylindersRet",
                          PT := T#2S);
   "alarm1".%X0 := "IEC_Timer_0_DB_9".Q OR (NOT "DB_HMI".alarmAckmowledge AND "alarm1".%X0);
END_REGION

REGION Network 18: 2.1 - INSERT EUCHNER KEY
   RUNG wire#powerrail
      Contact( "DB_HMI".insertAlarmKey )
      wire#w1
      Coil( "alarm1".%X1 )
   END_RUNG
   RUNG wire#powerrail
      I_Contact( "DB_HMI".alarmAckmowledge )
      Contact( "alarm1".%X1 )
   END_RUNG wire#w1
   RUNG wire#powerrail
      Contact( "DB_HMI".alarmAckmowledge )
      R_Coil( "DB_HMI".insertAlarmKey )
   END_RUNG
   // the same network as SCL:
   "alarm1".%X1 := "DB_HMI".insertAlarmKey OR (NOT "DB_HMI".alarmAckmowledge AND "alarm1".%X1);
   IF "DB_HMI".alarmAckmowledge THEN "DB_HMI".insertAlarmKey := FALSE; END_IF;
END_REGION

REGION Network 19: 2.2 - TORQUE NOK RESTART
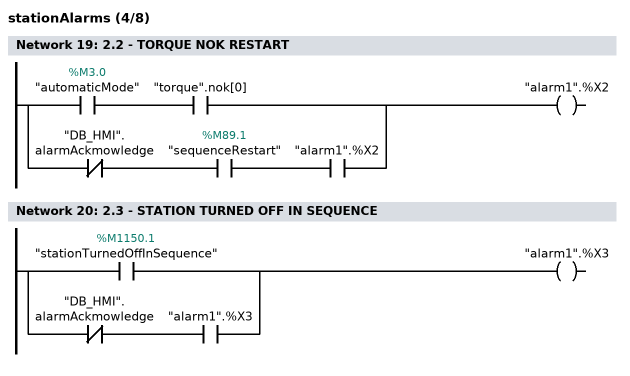
   RUNG wire#powerrail
      Contact( "automaticMode" )
      Contact( "torque".nok[0] )
      wire#w1
      Coil( "alarm1".%X2 )
   END_RUNG
   RUNG wire#powerrail
      I_Contact( "DB_HMI".alarmAckmowledge )
      Contact( "sequenceRestart" )
      Contact( "alarm1".%X2 )
   END_RUNG wire#w1
   // the same network as SCL:
   "alarm1".%X2 := ("automaticMode" AND "torque".nok[0]) OR (NOT "DB_HMI".alarmAckmowledge AND "sequenceRestart" AND "alarm1".%X2);
END_REGION

REGION Network 20: 2.3 - STATION TURNED OFF IN SEQUENCE
   RUNG wire#powerrail
      Contact( "stationTurnedOffInSequence" )
      wire#w1
      Coil( "alarm1".%X3 )
   END_RUNG
   RUNG wire#powerrail
      I_Contact( "DB_HMI".alarmAckmowledge )
      Contact( "alarm1".%X3 )
   END_RUNG wire#w1
   // the same network as SCL:
   "alarm1".%X3 := "stationTurnedOffInSequence" OR (NOT "DB_HMI".alarmAckmowledge AND "alarm1".%X3);
END_REGION

REGION Network 21: 2.4-2.13 - COMMUNICATION ALARMS
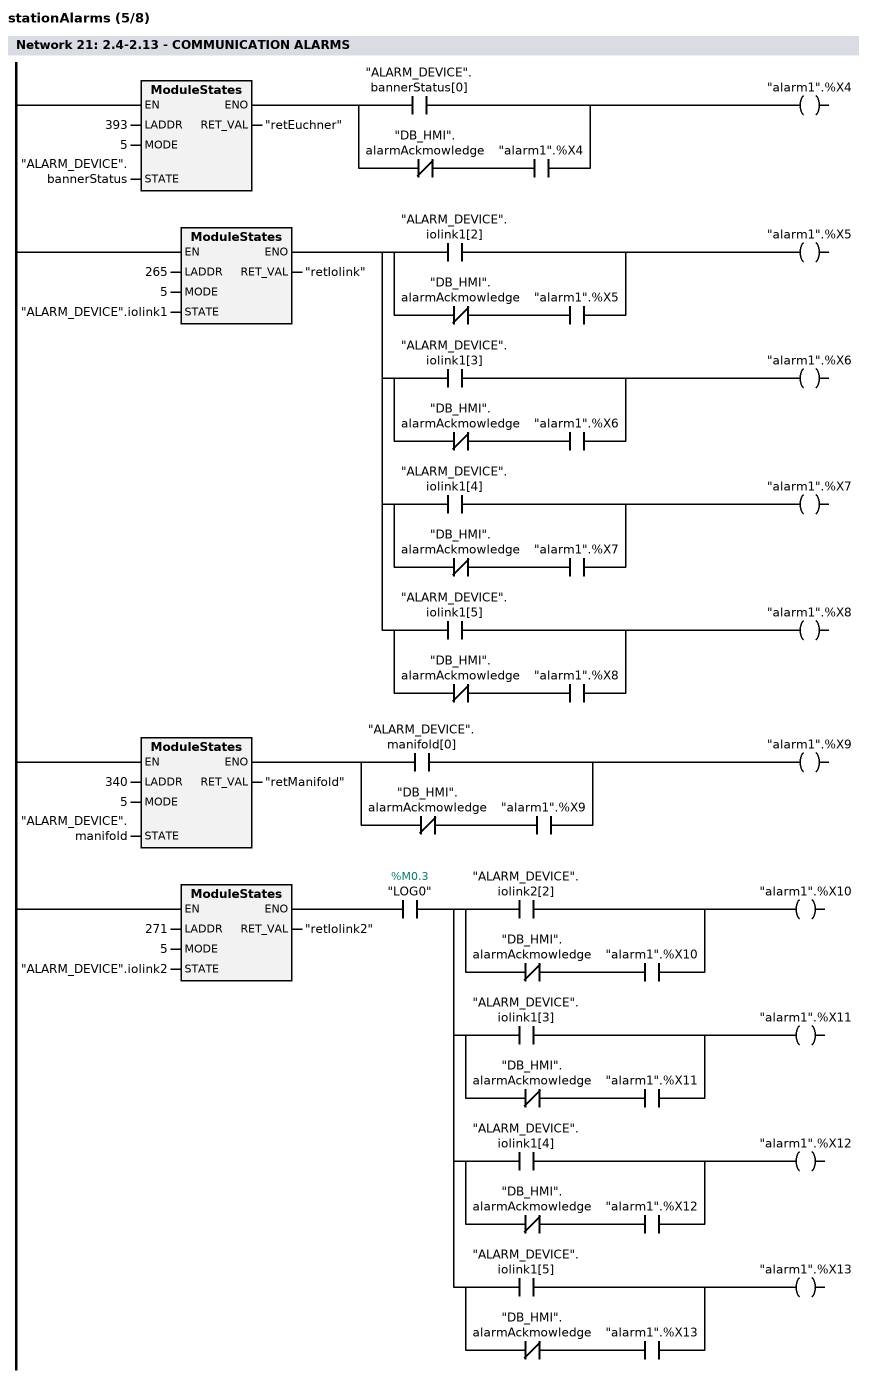
   RUNG wire#powerrail
      ModuleStates(LADDR := 393, MODE := 5, STATE := "ALARM_DEVICE".bannerStatus, Ret_Val => "retEuchner")
      wire#w1
      Contact( "ALARM_DEVICE".bannerStatus[0] )
      wire#w2
      Coil( "alarm1".%X4 )
   END_RUNG
   RUNG wire#w1
      I_Contact( "DB_HMI".alarmAckmowledge )
      Contact( "alarm1".%X4 )
   END_RUNG wire#w2
   RUNG wire#powerrail
      ModuleStates(LADDR := 265, MODE := 5, STATE := "ALARM_DEVICE".iolink1, Ret_Val => "retIolink")
      wire#w3
      Contact( "ALARM_DEVICE".iolink1[2] )
      wire#w4
      Coil( "alarm1".%X5 )
   END_RUNG
   RUNG wire#w3
      I_Contact( "DB_HMI".alarmAckmowledge )
      Contact( "alarm1".%X5 )
   END_RUNG wire#w4
   RUNG wire#w3
      Contact( "ALARM_DEVICE".iolink1[3] )
      wire#w5
      Coil( "alarm1".%X6 )
   END_RUNG
   RUNG wire#w3
      I_Contact( "DB_HMI".alarmAckmowledge )
      Contact( "alarm1".%X6 )
   END_RUNG wire#w5
   RUNG wire#w3
      Contact( "ALARM_DEVICE".iolink1[4] )
      wire#w6
      Coil( "alarm1".%X7 )
   END_RUNG
   RUNG wire#w3
      I_Contact( "DB_HMI".alarmAckmowledge )
      Contact( "alarm1".%X7 )
   END_RUNG wire#w6
   RUNG wire#w3
      Contact( "ALARM_DEVICE".iolink1[5] )
      wire#w7
      Coil( "alarm1".%X8 )
   END_RUNG
   RUNG wire#w3
      I_Contact( "DB_HMI".alarmAckmowledge )
      Contact( "alarm1".%X8 )
   END_RUNG wire#w7
   RUNG wire#powerrail
      ModuleStates(LADDR := 340, MODE := 5, STATE := "ALARM_DEVICE".manifold, Ret_Val => "retManifold")
      wire#w8
      Contact( "ALARM_DEVICE".manifold[0] )
      wire#w9
      Coil( "alarm1".%X9 )
   END_RUNG
   RUNG wire#w8
      I_Contact( "DB_HMI".alarmAckmowledge )
      Contact( "alarm1".%X9 )
   END_RUNG wire#w9
   RUNG wire#powerrail
      ModuleStates(LADDR := 271, MODE := 5, STATE := "ALARM_DEVICE".iolink2, Ret_Val => "retIolink2")
      Contact( "LOG0" )
      wire#w10
      Contact( "ALARM_DEVICE".iolink2[2] )
      wire#w11
      Coil( "alarm1".%X10 )
   END_RUNG
   RUNG wire#w10
      I_Contact( "DB_HMI".alarmAckmowledge )
      Contact( "alarm1".%X10 )
   END_RUNG wire#w11
   RUNG wire#w10
      Contact( "ALARM_DEVICE".iolink1[3] )
      wire#w12
      Coil( "alarm1".%X11 )
   END_RUNG
   RUNG wire#w10
      I_Contact( "DB_HMI".alarmAckmowledge )
      Contact( "alarm1".%X11 )
   END_RUNG wire#w12
   RUNG wire#w10
      Contact( "ALARM_DEVICE".iolink1[4] )
      wire#w13
      Coil( "alarm1".%X12 )
   END_RUNG
   RUNG wire#w10
      I_Contact( "DB_HMI".alarmAckmowledge )
      Contact( "alarm1".%X12 )
   END_RUNG wire#w13
   RUNG wire#w10
      Contact( "ALARM_DEVICE".iolink1[5] )
      wire#w14
      Coil( "alarm1".%X13 )
   END_RUNG
   RUNG wire#w10
      I_Contact( "DB_HMI".alarmAckmowledge )
      Contact( "alarm1".%X13 )
   END_RUNG wire#w14
   // the same network as SCL:
   "retEuchner" := ModuleStates(LADDR := 393, MODE := 5, STATE := "ALARM_DEVICE".bannerStatus, ENO => #_w1);
   "alarm1".%X4 := #_w1 AND ("ALARM_DEVICE".bannerStatus[0] OR (NOT "DB_HMI".alarmAckmowledge AND "alarm1".%X4));
   "retIolink" := ModuleStates(LADDR := 265, MODE := 5, STATE := "ALARM_DEVICE".iolink1, ENO => #_w2);
   "alarm1".%X5 := #_w2 AND ("ALARM_DEVICE".iolink1[2] OR (NOT "DB_HMI".alarmAckmowledge AND "alarm1".%X5));
   "alarm1".%X6 := #_w2 AND ("ALARM_DEVICE".iolink1[3] OR (NOT "DB_HMI".alarmAckmowledge AND "alarm1".%X6));
   "alarm1".%X7 := #_w2 AND ("ALARM_DEVICE".iolink1[4] OR (NOT "DB_HMI".alarmAckmowledge AND "alarm1".%X7));
   "alarm1".%X8 := #_w2 AND ("ALARM_DEVICE".iolink1[5] OR (NOT "DB_HMI".alarmAckmowledge AND "alarm1".%X8));
   "retManifold" := ModuleStates(LADDR := 340, MODE := 5, STATE := "ALARM_DEVICE".manifold, ENO => #_w3);
   "alarm1".%X9 := #_w3 AND ("ALARM_DEVICE".manifold[0] OR (NOT "DB_HMI".alarmAckmowledge AND "alarm1".%X9));
   "retIolink2" := ModuleStates(LADDR := 271, MODE := 5, STATE := "ALARM_DEVICE".iolink2, ENO => #_w4);
   #_w5 := #_w4 AND "LOG0";
   "alarm1".%X10 := #_w5 AND ("ALARM_DEVICE".iolink2[2] OR (NOT "DB_HMI".alarmAckmowledge AND "alarm1".%X10));
   "alarm1".%X11 := #_w5 AND ("ALARM_DEVICE".iolink1[3] OR (NOT "DB_HMI".alarmAckmowledge AND "alarm1".%X11));
   "alarm1".%X12 := #_w5 AND ("ALARM_DEVICE".iolink1[4] OR (NOT "DB_HMI".alarmAckmowledge AND "alarm1".%X12));
   "alarm1".%X13 := #_w5 AND ("ALARM_DEVICE".iolink1[5] OR (NOT "DB_HMI".alarmAckmowledge AND "alarm1".%X13));
END_REGION

REGION Network 22: 2.14.- TORQUE TO ACTIVATION POS
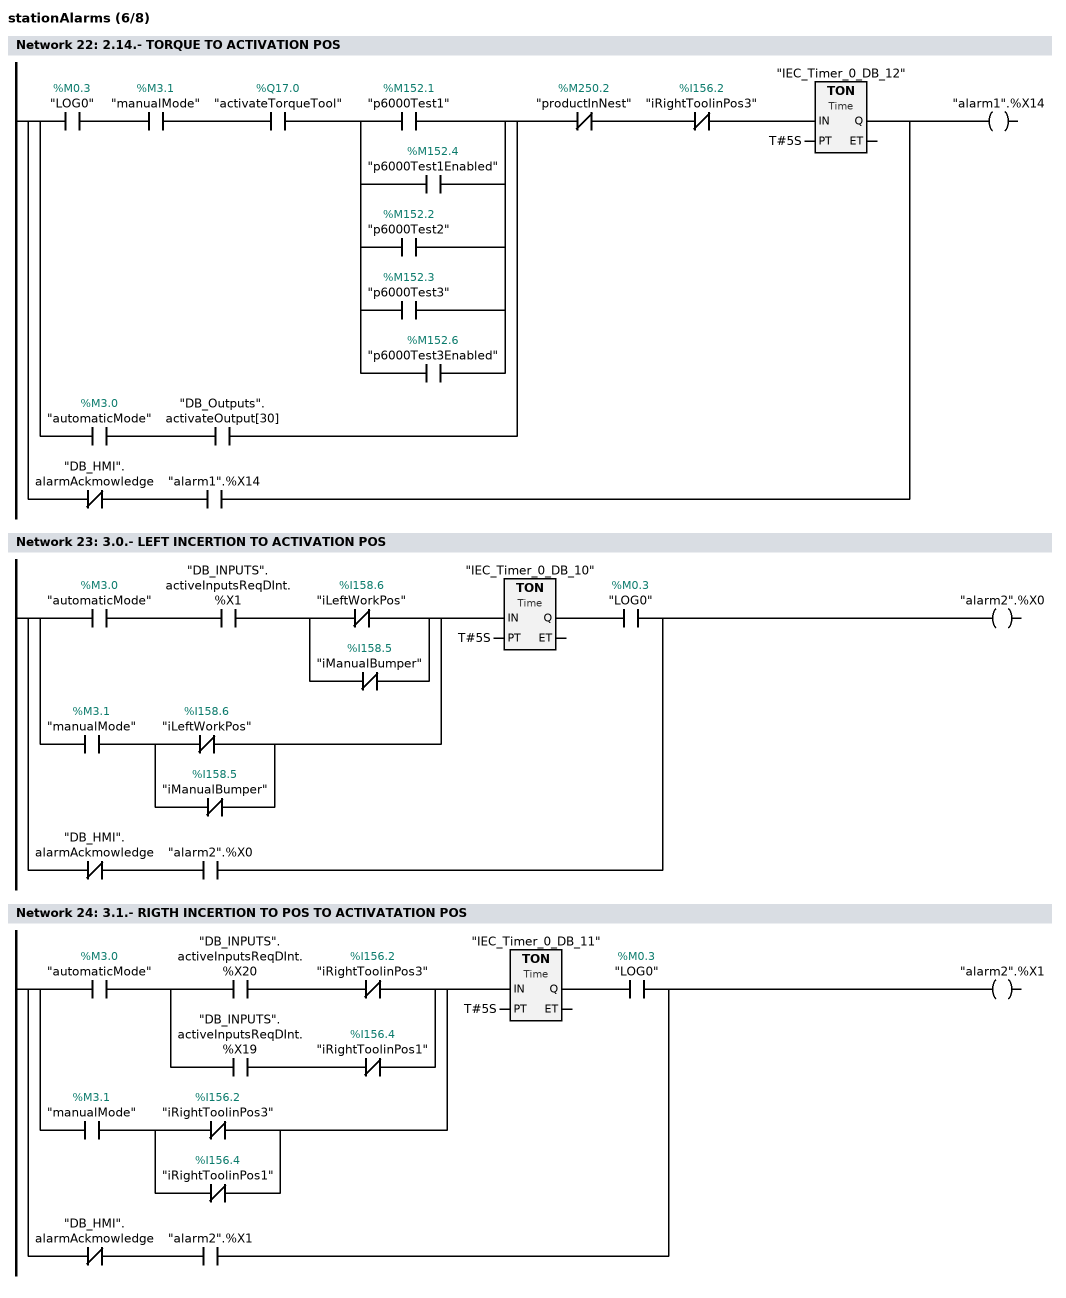
   RUNG wire#powerrail
      Contact( "LOG0" )
      Contact( "manualMode" )
      Contact( "activateTorqueTool" )
      wire#w1
      Contact( "p6000Test1" )
      wire#w2
      I_Contact( "productInNest" )
      I_Contact( "iRightToolinPos3" )
      { S7_Templates := "time_type := Time" } "IEC_Timer_0_DB_12".TON(pt := T#5S, et =>)
      wire#w3
      Coil( "alarm1".%X14 )
   END_RUNG
   RUNG wire#w1
      Contact( "p6000Test1Enabled" )
   END_RUNG wire#w2
   RUNG wire#w1
      Contact( "p6000Test2" )
   END_RUNG wire#w2
   RUNG wire#w1
      Contact( "p6000Test3" )
   END_RUNG wire#w2
   RUNG wire#w1
      Contact( "p6000Test3Enabled" )
   END_RUNG wire#w2
   RUNG wire#powerrail
      Contact( "automaticMode" )
      Contact( "DB_Outputs".activateOutput[30] )
   END_RUNG wire#w2
   RUNG wire#powerrail
      I_Contact( "DB_HMI".alarmAckmowledge )
      Contact( "alarm1".%X14 )
   END_RUNG wire#w3
   // the same network as SCL:
   "IEC_Timer_0_DB_12".TON(IN := (("LOG0" AND "manualMode" AND "activateTorqueTool" AND ("p6000Test1" OR "p6000Test1Enabled" OR "p6000Test2" OR "p6000Test3" OR "p6000Test3Enabled")) OR ("automaticMode" AND "DB_Outputs".activateOutput[30])) AND NOT "productInNest" AND NOT "iRightToolinPos3",
                           PT := T#5S);
   "alarm1".%X14 := "IEC_Timer_0_DB_12".Q OR (NOT "DB_HMI".alarmAckmowledge AND "alarm1".%X14);
END_REGION

REGION Network 23: 3.0.- LEFT INCERTION TO ACTIVATION POS
   RUNG wire#powerrail
      Contact( "automaticMode" )
      Contact( "DB_INPUTS".activeInputsReqDInt.%X1 )
      wire#w1
      I_Contact( "iLeftWorkPos" )
      wire#w2
      { S7_Templates := "time_type := Time" } "IEC_Timer_0_DB_10".TON(pt := T#5S, et =>)
      Contact( "LOG0" )
      wire#w4
      Coil( "alarm2".%X0 )
   END_RUNG
   RUNG wire#w1
      I_Contact( "iManualBumper" )
   END_RUNG wire#w2
   RUNG wire#powerrail
      Contact( "manualMode" )
      wire#w3
      I_Contact( "iLeftWorkPos" )
   END_RUNG wire#w2
   RUNG wire#w3
      I_Contact( "iManualBumper" )
   END_RUNG wire#w2
   RUNG wire#powerrail
      I_Contact( "DB_HMI".alarmAckmowledge )
      Contact( "alarm2".%X0 )
   END_RUNG wire#w4
   // the same network as SCL:
   "IEC_Timer_0_DB_10".TON(IN := ("automaticMode" AND "DB_INPUTS".activeInputsReqDInt.%X1 AND (NOT "iLeftWorkPos" OR NOT "iManualBumper")) OR ("manualMode" AND (NOT "iLeftWorkPos" OR NOT "iManualBumper")),
                           PT := T#5S);
   "alarm2".%X0 := ("IEC_Timer_0_DB_10".Q AND "LOG0") OR (NOT "DB_HMI".alarmAckmowledge AND "alarm2".%X0);
END_REGION

REGION Network 24: 3.1.- RIGTH INCERTION TO POS TO ACTIVATATION POS
   RUNG wire#powerrail
      Contact( "automaticMode" )
      wire#w1
      Contact( "DB_INPUTS".activeInputsReqDInt.%X20 )
      I_Contact( "iRightToolinPos3" )
      wire#w2
      { S7_Templates := "time_type := Time" } "IEC_Timer_0_DB_11".TON(pt := T#5S, et =>)
      Contact( "LOG0" )
      wire#w4
      Coil( "alarm2".%X1 )
   END_RUNG
   RUNG wire#w1
      Contact( "DB_INPUTS".activeInputsReqDInt.%X19 )
      I_Contact( "iRightToolinPos1" )
   END_RUNG wire#w2
   RUNG wire#powerrail
      Contact( "manualMode" )
      wire#w3
      I_Contact( "iRightToolinPos3" )
   END_RUNG wire#w2
   RUNG wire#w3
      I_Contact( "iRightToolinPos1" )
   END_RUNG wire#w2
   RUNG wire#powerrail
      I_Contact( "DB_HMI".alarmAckmowledge )
      Contact( "alarm2".%X1 )
   END_RUNG wire#w4
   // the same network as SCL:
   "IEC_Timer_0_DB_11".TON(IN := ("automaticMode" AND (("DB_INPUTS".activeInputsReqDInt.%X20 AND NOT "iRightToolinPos3") OR ("DB_INPUTS".activeInputsReqDInt.%X19 AND NOT "iRightToolinPos1"))) OR ("manualMode" AND (NOT "iRightToolinPos3" OR NOT "iRightToolinPos1")),
                           PT := T#5S);
   "alarm2".%X1 := ("IEC_Timer_0_DB_11".Q AND "LOG0") OR (NOT "DB_HMI".alarmAckmowledge AND "alarm2".%X1);
END_REGION

REGION Network 25: 3.2.- POWER TOOLING NOT CONNECTED
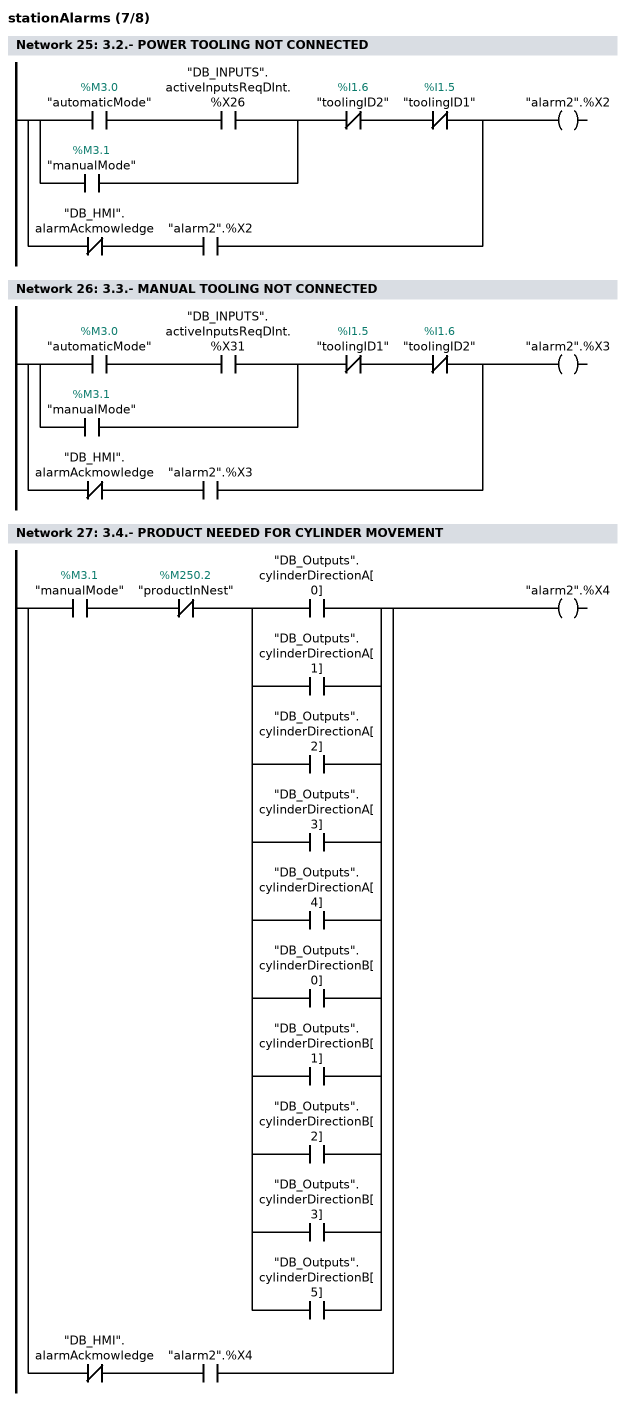
   RUNG wire#powerrail
      Contact( "automaticMode" )
      Contact( "DB_INPUTS".activeInputsReqDInt.%X26 )
      wire#w1
      I_Contact( "toolingID2" )
      I_Contact( "toolingID1" )
      wire#w2
      Coil( "alarm2".%X2 )
   END_RUNG
   RUNG wire#powerrail
      Contact( "manualMode" )
   END_RUNG wire#w1
   RUNG wire#powerrail
      I_Contact( "DB_HMI".alarmAckmowledge )
      Contact( "alarm2".%X2 )
   END_RUNG wire#w2
   // the same network as SCL:
   "alarm2".%X2 := ((("automaticMode" AND "DB_INPUTS".activeInputsReqDInt.%X26) OR "manualMode") AND NOT "toolingID2" AND NOT "toolingID1") OR (NOT "DB_HMI".alarmAckmowledge AND "alarm2".%X2);
END_REGION

REGION Network 26: 3.3.- MANUAL TOOLING NOT CONNECTED
   RUNG wire#powerrail
      Contact( "automaticMode" )
      Contact( "DB_INPUTS".activeInputsReqDInt.%X31 )
      wire#w1
      I_Contact( "toolingID1" )
      I_Contact( "toolingID2" )
      wire#w2
      Coil( "alarm2".%X3 )
   END_RUNG
   RUNG wire#powerrail
      Contact( "manualMode" )
   END_RUNG wire#w1
   RUNG wire#powerrail
      I_Contact( "DB_HMI".alarmAckmowledge )
      Contact( "alarm2".%X3 )
   END_RUNG wire#w2
   // the same network as SCL:
   "alarm2".%X3 := ((("automaticMode" AND "DB_INPUTS".activeInputsReqDInt.%X31) OR "manualMode") AND NOT "toolingID1" AND NOT "toolingID2") OR (NOT "DB_HMI".alarmAckmowledge AND "alarm2".%X3);
END_REGION

REGION Network 27: 3.4.- PRODUCT NEEDED FOR CYLINDER MOVEMENT
   RUNG wire#powerrail
      Contact( "manualMode" )
      I_Contact( "productInNest" )
      wire#w1
      Contact( "DB_Outputs".cylinderDirectionA[0] )
      wire#w2
      Coil( "alarm2".%X4 )
   END_RUNG
   RUNG wire#w1
      Contact( "DB_Outputs".cylinderDirectionA[1] )
   END_RUNG wire#w2
   RUNG wire#w1
      Contact( "DB_Outputs".cylinderDirectionA[2] )
   END_RUNG wire#w2
   RUNG wire#w1
      Contact( "DB_Outputs".cylinderDirectionA[3] )
   END_RUNG wire#w2
   RUNG wire#w1
      Contact( "DB_Outputs".cylinderDirectionA[4] )
   END_RUNG wire#w2
   RUNG wire#w1
      Contact( "DB_Outputs".cylinderDirectionB[0] )
   END_RUNG wire#w2
   RUNG wire#w1
      Contact( "DB_Outputs".cylinderDirectionB[1] )
   END_RUNG wire#w2
   RUNG wire#w1
      Contact( "DB_Outputs".cylinderDirectionB[2] )
   END_RUNG wire#w2
   RUNG wire#w1
      Contact( "DB_Outputs".cylinderDirectionB[3] )
   END_RUNG wire#w2
   RUNG wire#w1
      Contact( "DB_Outputs".cylinderDirectionB[5] )
   END_RUNG wire#w2
   RUNG wire#powerrail
      I_Contact( "DB_HMI".alarmAckmowledge )
      Contact( "alarm2".%X4 )
   END_RUNG wire#w2
   // the same network as SCL:
   "alarm2".%X4 := ("manualMode" AND NOT "productInNest" AND ("DB_Outputs".cylinderDirectionA[0] OR "DB_Outputs".cylinderDirectionA[1] OR "DB_Outputs".cylinderDirectionA[2] OR "DB_Outputs".cylinderDirectionA[3] OR "DB_Outputs".cylinderDirectionA[4] OR "DB_Outputs".cylinderDirectionB[0] OR "DB_Outputs".cylinderDirectionB[1] OR "DB_Outputs".cylinderDirectionB[2] OR "DB_Outputs".cylinderDirectionB[3] OR "DB_Outputs".cylinderDirectionB[5])) OR (NOT "DB_HMI".alarmAckmowledge AND "alarm2".%X4);
END_REGION

REGION Network 28: 3.5.- MAN LH PROD NOK ROD
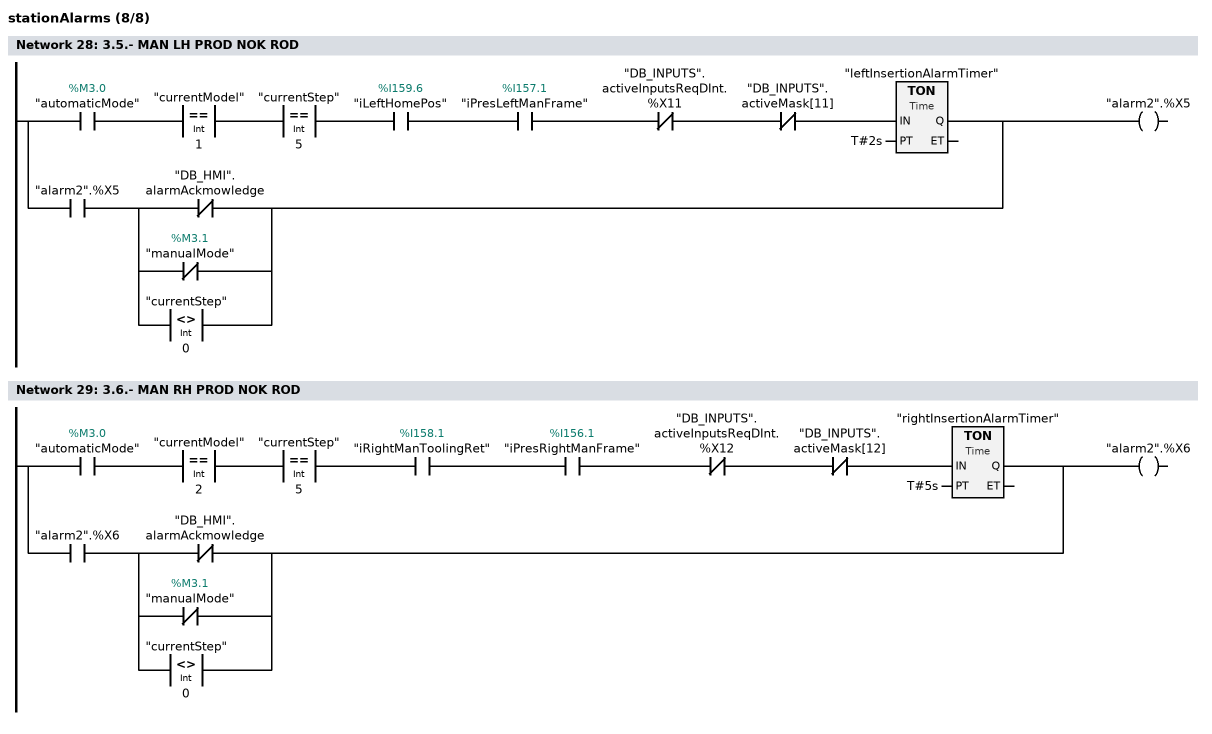
   RUNG wire#powerrail
      Contact( "automaticMode" )
      { S7_Templates := "SrcType := Int" } EQ_Contact(in1 := "currentModel", in2 := 1)
      { S7_Templates := "SrcType := Int" } EQ_Contact(in1 := "currentStep", in2 := 5)
      Contact( "iLeftHomePos" )
      Contact( "iPresLeftManFrame" )
      I_Contact( "DB_INPUTS".activeInputsReqDInt.%X11 )
      I_Contact( "DB_INPUTS".activeMask[11] )
      { S7_Templates := "time_type := Time" } "leftInsertionAlarmTimer".TON(pt := T#2s, et =>)
      wire#w1
      Coil( "alarm2".%X5 )
   END_RUNG
   RUNG wire#powerrail
      Contact( "alarm2".%X5 )
      wire#w2
      I_Contact( "DB_HMI".alarmAckmowledge )
   END_RUNG wire#w1
   RUNG wire#w2
      I_Contact( "manualMode" )
   END_RUNG wire#w1
   RUNG wire#w2
      { S7_Templates := "SrcType := Int" } NE_Contact(in1 := "currentStep", in2 := 0)
   END_RUNG wire#w1
   // the same network as SCL:
   "leftInsertionAlarmTimer".TON(IN := "automaticMode" AND ("currentModel" = 1) AND ("currentStep" = 5) AND "iLeftHomePos" AND "iPresLeftManFrame" AND NOT "DB_INPUTS".activeInputsReqDInt.%X11 AND NOT "DB_INPUTS".activeMask[11],
                           PT := T#2s);
   "alarm2".%X5 := "leftInsertionAlarmTimer".Q OR ("alarm2".%X5 AND (NOT "DB_HMI".alarmAckmowledge OR NOT "manualMode" OR ("currentStep" <> 0)));
END_REGION

REGION Network 29: 3.6.- MAN RH PROD NOK ROD
   RUNG wire#powerrail
      Contact( "automaticMode" )
      { S7_Templates := "SrcType := Int" } EQ_Contact(in1 := "currentModel", in2 := 2)
      { S7_Templates := "SrcType := Int" } EQ_Contact(in1 := "currentStep", in2 := 5)
      Contact( "iRightManToolingRet" )
      Contact( "iPresRightManFrame" )
      I_Contact( "DB_INPUTS".activeInputsReqDInt.%X12 )
      I_Contact( "DB_INPUTS".activeMask[12] )
      { S7_Templates := "time_type := Time" } "rightInsertionAlarmTimer".TON(pt := T#5s, et =>)
      wire#w1
      Coil( "alarm2".%X6 )
   END_RUNG
   RUNG wire#powerrail
      Contact( "alarm2".%X6 )
      wire#w2
      I_Contact( "DB_HMI".alarmAckmowledge )
   END_RUNG wire#w1
   RUNG wire#w2
      I_Contact( "manualMode" )
   END_RUNG wire#w1
   RUNG wire#w2
      { S7_Templates := "SrcType := Int" } NE_Contact(in1 := "currentStep", in2 := 0)
   END_RUNG wire#w1
   // the same network as SCL:
   "rightInsertionAlarmTimer".TON(IN := "automaticMode" AND ("currentModel" = 2) AND ("currentStep" = 5) AND "iRightManToolingRet" AND "iPresRightManFrame" AND NOT "DB_INPUTS".activeInputsReqDInt.%X12 AND NOT "DB_INPUTS".activeMask[12],
                           PT := T#5s);
   "alarm2".%X6 := "rightInsertionAlarmTimer".Q OR ("alarm2".%X6 AND (NOT "DB_HMI".alarmAckmowledge OR NOT "manualMode" OR ("currentStep" <> 0)));
END_REGION
END_FUNCTION

FUNCTION "production" : Void   // FC15, LAD
{ S7_Optimized_Access := 'TRUE' }
VERSION : 0.1
// stored: AutoNumber true, IsIECCheckEnabled false, SetENOAutomatically false, UDAEnableTagReadback false
   VAR_TEMP   // added for the SCL form of the ladder/FBD networks
      _w1 : Bool;
      _w2 : Bool;
      _w3 : Bool;
   END_VAR
BEGIN

REGION Network 1: SHIFTS PRODUCTION
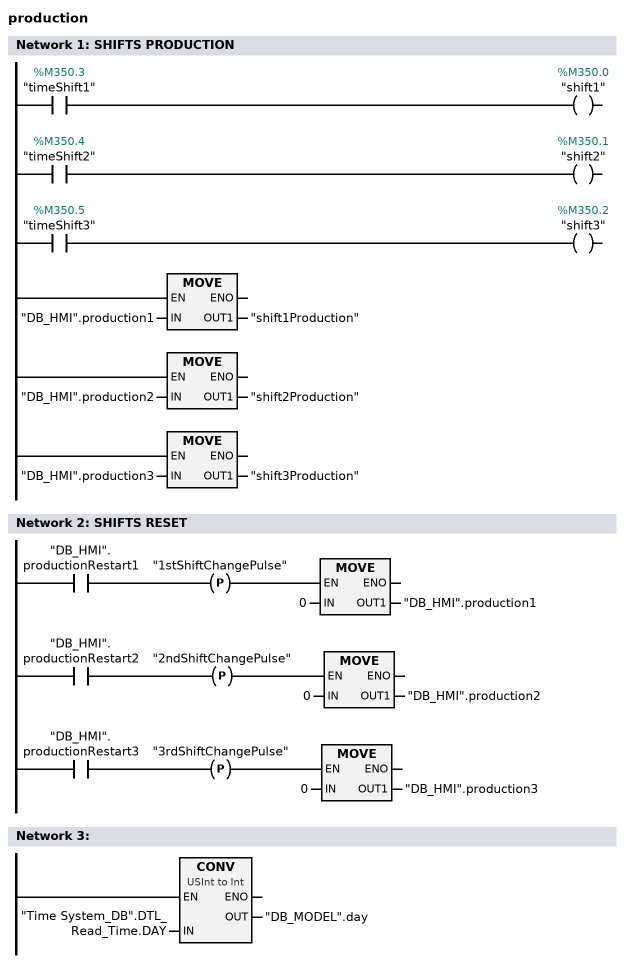
   RUNG wire#powerrail
      Contact( "timeShift1" )
      Coil( "shift1" )
   END_RUNG
   RUNG wire#powerrail
      Contact( "timeShift2" )
      Coil( "shift2" )
   END_RUNG
   RUNG wire#powerrail
      Contact( "timeShift3" )
      Coil( "shift3" )
   END_RUNG
   RUNG wire#powerrail
      Move(in := "DB_HMI".production1, out1 => "shift1Production")
   END_RUNG
   RUNG wire#powerrail
      Move(in := "DB_HMI".production2, out1 => "shift2Production")
   END_RUNG
   RUNG wire#powerrail
      Move(in := "DB_HMI".production3, out1 => "shift3Production")
   END_RUNG
   // the same network as SCL:
   "shift1" := "timeShift1";
   "shift2" := "timeShift2";
   "shift3" := "timeShift3";
   "shift1Production" := "DB_HMI".production1;
   "shift2Production" := "DB_HMI".production2;
   "shift3Production" := "DB_HMI".production3;
END_REGION

REGION Network 2: SHIFTS RESET
   RUNG wire#powerrail
      Contact( "DB_HMI".productionRestart1 )
      P_Trig( "1stShiftChangePulse" )
      Move(in := 0, out1 => "DB_HMI".production1)
   END_RUNG
   RUNG wire#powerrail
      Contact( "DB_HMI".productionRestart2 )
      P_Trig( "2ndShiftChangePulse" )
      Move(in := 0, out1 => "DB_HMI".production2)
   END_RUNG
   RUNG wire#powerrail
      Contact( "DB_HMI".productionRestart3 )
      P_Trig( "3rdShiftChangePulse" )
      Move(in := 0, out1 => "DB_HMI".production3)
   END_RUNG
   // the same network as SCL:
   #_w1 := "DB_HMI".productionRestart1 AND NOT "1stShiftChangePulse";   // rising edge
   "1stShiftChangePulse" := "DB_HMI".productionRestart1;
   IF #_w1 THEN "DB_HMI".production1 := 0; END_IF;
   #_w2 := "DB_HMI".productionRestart2 AND NOT "2ndShiftChangePulse";   // rising edge
   "2ndShiftChangePulse" := "DB_HMI".productionRestart2;
   IF #_w2 THEN "DB_HMI".production2 := 0; END_IF;
   #_w3 := "DB_HMI".productionRestart3 AND NOT "3rdShiftChangePulse";   // rising edge
   "3rdShiftChangePulse" := "DB_HMI".productionRestart3;
   IF #_w3 THEN "DB_HMI".production3 := 0; END_IF;
END_REGION

REGION Network 3
   RUNG wire#powerrail
      { S7_Templates := "[SrcType := USInt, DestType := Int]" } Convert(in := "Time System_DB".DTL_Read_Time.DAY, out => "DB_MODEL".day)
   END_RUNG
   // the same network as SCL:
   "DB_MODEL".day := USINT_TO_INT("Time System_DB".DTL_Read_Time.DAY);
END_REGION
END_FUNCTION

FUNCTION_BLOCK "Time System"   // FB2420, LAD
{ S7_Optimized_Access := 'TRUE' }
VERSION : 0.1
// stored: AutoNumber false, IsIECCheckEnabled false, IsRetainMemResEnabled false, MemoryReserve 100, SetENOAutomatically false, UDAEnableTagReadback false
   VAR_INPUT
      bPartOkNok : Bool;
      bRunningcycle : Bool;
      bPreCount : Bool;
   END_VAR
   VAR_OUTPUT
      bShift1 : Bool;
      bShift2 : Bool;
      bShift3 : Bool;
      nCycle_Time_Shift : Real;
      nCycleTimeAvg_Shift1 : Real;
      nCycleTimeAvg_Shift2 : Real;
      nCycleTimeAvg_Shift3 : Real;
   END_VAR
   VAR
      Ret_Val_WR { ExternalAccessible := 'False'; ExternalVisible := 'False'; ExternalWritable := 'False'} : USInt;
      Ret_Val_RD { ExternalAccessible := 'False'; ExternalVisible := 'False'; ExternalWritable := 'False'} : USInt;
      DTL_Set_Time : DTL;
      DTL_Read_Time : DTL;
      TOD_Read : Time_Of_Day;
      Date_Read : Date;
      bAceptButtonHmiP : Bool;
      bAcept_buttonHMI : Bool;
      nSet_minute : Int;
      nSet_Hour : Int;
      nSet_Day : Int;
      nSet_Month : Int;
      nSet_Year : Int;
      nCycleTimeArray : Array[0..5] of Real;
      tCycleTime { S7_SetPoint := 'True'} : IEC_TIMER;
      nCycleTimeET : UDInt;
      tCycleTimeTotal : UDInt;
      bPartOkNokP : Bool;
      bPartOkNokCmd : Bool;
      nPartAvgCounter : Int;
      bCycle_StartedP : Bool;
      bSH1 : Bool;
      bSH2 : Bool;
      bSH3 : Bool;
      nCycle_Time : Real;
      nCycleTimeAvg : Real;
      Read_Local_Time : DTL;
      Read_System_Time : DTL;
      Time_HMI_Set : DTL;
      RetVal1 : Word;
      Retval2 : Word;
      Retval3 : Word;
      n : Int;
      timesCounter { S7_SetPoint := 'True'} : IEC_COUNTER;
   END_VAR
   VAR RETAIN
      tCycle_Running : Real;
   END_VAR
   VAR
      nCycleAvg : DInt;
      nCycleTime_Total : Time_Of_Day;
      ntimeRun_conv : UDInt;
   END_VAR
   // nCycleTimeArray[3..5] := 0.0;
   VAR_TEMP   // added for the SCL form of the ladder/FBD networks
      _w1 : Bool;
   END_VAR
BEGIN

REGION Network 1: SET HOUR
